FUNCTION_BLOCK FB 1051
TITLE = Blower PMP01
//Creation:
//Date:            Author:                                               Version
//--------------------------------------------------------------------------------
//29.03.2018     ilia                                   01.00.00
//
//Changes:
//No. Date:        Who       Description                           Mark   Version 
//--------------------------------------------------------------------------------
//01
//________________________________________________________________________________
//Function:
//1. Maximum 6 switching cycles per hour ' 10 minutes restart protection time
//
AUTHOR : ilia
NAME : project
VERSION : 1.0
VAR_INPUT
  IF_VP1_FC_DB : INT ;
  IF_VP1_FC_DW : INT ;
  i_piwPressureVP1 : INT ;	//analogue input address
  i_xSystemActive : BOOL ;	//system control on
  i_xFAValveClose : BOOL ;
  i_xFAValveOpen : BOOL ;
  ack_xFAValve : BOOL ;
  ack_OverPressureVP1 : BOOL ;
END_VAR
VAR_IN_OUT
  q_xFAValve : BOOL ;	//Fresh Air ventil
  f_xFAValve : BOOL ;	//Fault fresh air ventil
  f_xPressureFaultVP01 : BOOL ;	//Pressure Fault
  f_xBrokenWireVP01 : BOOL ;	//Broken wire pressure fault
  f_xParErrorVP01 : BOOL ;	//False parameter pressure transmitter
END_VAR
VAR
  reserve_IO : ARRAY  [10 .. 49 ] OF BYTE ;
  HMI : STRUCT 	//Interface of HMI
   CMD : STRUCT
    reserve : BOOL ;
    reserve_1 : BOOL ;
    reserve_2 : BOOL ;
    reserve_3 : BOOL ;
    reserve_4 : BOOL ;
    reserve_5 : BOOL ;
    reserve_6 : BOOL ;
    reserve_7 : BOOL ;
    reserve_8 : BOOL ;
    reserve_9 : BOOL ;
    reserve_10 : BOOL ;
    reserve_11 : BOOL ;
    reserve_12 : BOOL ;
    reserve_13 : BOOL ;
    reserve_14 : BOOL ;
    reserve_15 : BOOL ;
   END_STRUCT ;
   STATE : STRUCT
    xxPressureFault : BOOL ;
    xxEmtyPressure : BOOL ;
    xVP1Locked : BOOL ;
    reserve_4 : BOOL ;
    reserve_5 : BOOL ;
    reserve_6 : BOOL ;
    reserve_7 : BOOL ;
    reserve_8 : BOOL ;
    reserve_9 : BOOL ;
    reserve_10 : BOOL ;
    reserve_11 : BOOL ;
    reserve_12 : BOOL ;
    reserve_13 : BOOL ;
    reserve : BOOL ;
   END_STRUCT ;
   PARAM : STRUCT
    rOffDelayVPTime : REAL  := 6.000000e+001;
    rOnDelayHDTime : REAL ;
    res_1 : REAL ;
    res_2 : REAL ;
    res_3 : REAL ;
    res_4 : REAL  := 2.000000e+000;
    reserve_2 : REAL ;
    reserve_3 : REAL ;
    reserve_4 : INT ;
    reserve_4_1 : INT  := 6;
    reserve_6 : INT ;
    reserve_7 : INT ;
    reserve_8 : INT ;
    reserve_9 : INT ;
    reserve_9_1 : INT ;
   END_STRUCT ;
   PV : STRUCT
    rOffDelayVPTime : REAL ;
    rOnDelayHD : REAL ;
    rOffDelayRestart : REAL ;
    res : REAL ;
    res_1 : REAL ;
    res_2 : REAL ;
    res_3 : REAL ;
    res_4 : REAL ;
    reserve_4 : REAL ;
    reserve_8 : INT ;
    reserve_9 : INT ;
    reserve_10 : INT ;
    reserve_11 : INT ;
    reserve_8_1 : INT ;
   END_STRUCT ;
  END_STRUCT ;
  reserve_HMI : ARRAY  [146 .. 199 ] OF BYTE ;
  PROD : STRUCT 	//Interface of Production
   FROM : STRUCT
    reserve : INT ;
    reserve_1 : INT ;
    reserve_2 : INT ;
    reserve_3 : INT ;
    reserve_4 : INT ;
    reserve_5 : REAL ;
    reserve_6 : REAL ;
    CMD : STRUCT
     reserve : BOOL ;
     reserve_1 : BOOL ;
     reserve_2 : BOOL ;
     reserve_3 : BOOL ;
     reserve_4 : BOOL ;
     reserve_5 : BOOL ;
     reserve_6 : BOOL ;
     reserve_7 : BOOL ;
     reserve_8 : BOOL ;
     reserve_9 : BOOL ;
     reserve_10 : BOOL ;
     reserve_11 : BOOL ;
     reserve_12 : BOOL ;
     reserve_13 : BOOL ;
     reserve_14 : BOOL ;
     reserve_15 : BOOL ;
    END_STRUCT ;
   END_STRUCT ;
   TO : STRUCT
    reserve : INT ;
    reserve_1 : INT ;
    reserve_2 : INT ;
    reserve_3 : INT ;
    reserve_4 : INT ;
    reserve_5 : REAL ;
    reserve_6 : REAL ;
    STATE : STRUCT
     reserve : BOOL ;
     reserve_1 : BOOL ;
     reserve_2 : BOOL ;
     reserve_3 : BOOL ;
     reserve_4 : BOOL ;
     reserve_5 : BOOL ;
     reserve_6 : BOOL ;
     reserve_7 : BOOL ;
     reserve_8 : BOOL ;
     reserve_9 : BOOL ;
     reserve_10 : BOOL ;
     reserve_11 : BOOL ;
     reserve_12 : BOOL ;
     reserve_13 : BOOL ;
     reserve_14 : BOOL ;
     reserve_15 : BOOL ;
    END_STRUCT ;
   END_STRUCT ;
   reserve : ARRAY  [40 .. 49 ] OF BYTE ;
  END_STRUCT ;
  IF_Consumer : STRUCT 	//Interface Blower in blower object
   CONTROL : STRUCT
    Answer_DB : INT ;
    Answer_DW : INT ;
    iSpeedVP : INT ;
    reserve : INT ;
    reserve_3 : INT ;
    reserve_4 : REAL ;
    reserve_5 : REAL ;
    CMD : STRUCT
     xRequest : BOOL ;
     xRelease : BOOL ;
     reserve : BOOL ;
     reserve_1 : BOOL ;
     reserve_2 : BOOL ;
     reserve_3 : BOOL ;
     reserve_4 : BOOL ;
     reserve_5 : BOOL ;
     reserve_6 : BOOL ;
     reserve_7 : BOOL ;
     reserve_8 : BOOL ;
     reserve_9 : BOOL ;
     reserve_10 : BOOL ;
     reserve_11 : BOOL ;
     reserve_12 : BOOL ;
     reserve_13 : BOOL ;
    END_STRUCT ;
   END_STRUCT ;
   STATUS : STRUCT
    reserve_1 : INT ;
    reserve_2 : INT ;
    reserve_3 : INT ;
    reserve_4 : INT ;
    reserve_5 : INT ;
    rActualPressure : REAL ;
    reserve_6 : REAL ;
    STATE : STRUCT
     xReady : BOOL ;
     xActive : BOOL ;
     xPressureFault : BOOL ;
     xEmptyPressue : BOOL ;
     xFault : BOOL ;
     reserve : BOOL ;
     reserve_2 : BOOL ;
     reserve_3 : BOOL ;
     reserve_4 : BOOL ;
     reserve_5 : BOOL ;
     reserve_6 : BOOL ;
     reserve_7 : BOOL ;
     reserve_8 : BOOL ;
     reserve_9 : BOOL ;
     reserve_10 : BOOL ;
     reserve_11 : BOOL ;
    END_STRUCT ;
   END_STRUCT ;
  END_STRUCT ;
  IF_FC_VP1 : STRUCT 	//Interface FC in active object
   STATUS : STRUCT
    ActualFrequency : REAL ;
    reserve : INT ;
    reserve_1 : INT ;
    reserve_2 : INT ;
    reserve_3 : INT ;
    reserve_4 : INT ;
    reserve_5 : REAL ;
    STATE : STRUCT
     Ready : BOOL ;
     Active : BOOL ;
     Fault : BOOL ;
     reserve : BOOL ;
     reserve_1 : BOOL ;
     reserve_2 : BOOL ;
     reserve_3 : BOOL ;
     reserve_4 : BOOL ;
     reserve_5 : BOOL ;
     reserve_6 : BOOL ;
     reserve_7 : BOOL ;
     reserve_8 : BOOL ;
     reserve_9 : BOOL ;
     reserve_10 : BOOL ;
     reserve_11 : BOOL ;
     reserve_12 : BOOL ;
    END_STRUCT ;
   END_STRUCT ;
   CONTROL : STRUCT
    Answer_DB : INT ;
    Answer_DW : INT ;
    Frequency_Set : REAL ;
    No_motor_data : INT ;
    reserve : INT ;
    reserve_1 : INT ;
    reserve_2 : REAL ;
    CMD : STRUCT
     Request : BOOL ;
     Release : BOOL ;
     Left_run : BOOL ;
     reserve : BOOL ;
     reserve_1 : BOOL ;
     reserve_2 : BOOL ;
     reserve_3 : BOOL ;
     reserve_4 : BOOL ;
     reserve_5 : BOOL ;
     reserve_6 : BOOL ;
     reserve_7 : BOOL ;
     reserve_8 : BOOL ;
     reserve_9 : BOOL ;
     reserve_10 : BOOL ;
     reserve_11 : BOOL ;
     reserve_12 : BOOL ;
    END_STRUCT ;
   END_STRUCT ;
  END_STRUCT ;
  reserve_IF : ARRAY  [330 .. 499 ] OF BYTE ;
  VP1 : STRUCT 	//motor object
   parameter : STRUCT
    motor_on : BOOL  := TRUE;	//activate motor structure
    clock_on : BOOL ;	//activate clock structure
    FC_on : BOOL  := TRUE;	//activate frequency converter structure
    hour_meter_on : BOOL ;	//activate hour meter
    reserve_4 : BOOL ;
    reserve_5 : BOOL ;
    reserve_6 : BOOL ;
    reserve_7 : BOOL ;
   END_STRUCT ;
   quit_motor : BOOL ;	//1 = quit motor on
   input_motor : BOOL ;	//1 = input motor on (return indication)
   motor_locked : BOOL ;	//1 = motor locked (in manual and auto mode) e.g. repair-/safety switch
   auto_mode_control : BOOL ;	//1 = release/control of motor in auto mode
   motor_in_operation : BOOL ;	//1 = signal motor in operation
   fault : BOOL ;	//1 = signal motor fault
   man_mode_to_SCADA : BOOL ;	//0 = Automatik Mode, 1 = Hand Mode
   man_mode_from_SCADA : BOOL ;	//0 = Automatik Mode, 1 = Hand Mode
   man_mode_control : BOOL ;	//1 = release/control of motor in manual mode (from SCADA)
   man_mode_locked : BOOL ;	//1 = change to manual mode locked, motor is in automatic use
   start_with_impulse : BOOL  := TRUE;	//1 = start cycle with impulse
   set_cycles_reached : BOOL ;	//1 = set number of cycles has been reached
   continous_clock : BOOL  := TRUE;	//1 = continous clock / 0 = set number of clocks
   simulation : BOOL ;	//1 = simulation of object
   release_clock : BOOL ;	//1 = release bit for clock FC
   quit_clock : BOOL ;	//quit for clock FC, if release_clock = TRUE
   set_time_fault : INT  := 5;	//fault evaluation time in seconds
   actual_time_fault : INT ;	//actual fault evaluation time in seconds
   impulse_time : REAL  := 5.000000e+000;	//impulse time for clock in seconds
   break_time : REAL  := 5.000000e+000;	//break time for clock in seconds
   time_counter : REAL ;	//time counter (elapsed time)
   set_cycles : INT ;	//number of clocks if not continous clock
   clock_counter : INT ;	//clock counter
   FCs : STRUCT 	//frequency converter
    FC_in_operation : BOOL ;	//1 = FU in Betrieb
    fault : BOOL ;	//1 = FC fault
    set_revolutions_man_mode : INT  := 200;	//revolutions in permille in manual mode
    actual_revolutions : INT ;	//actual revolutions FC in man/auto mode
   END_STRUCT ;
   hour_meter : STRUCT 	//hour meter
    reset : BOOL ;	//reset hour meter
    warning : BOOL ;	//warning time exceeded
    alarm : BOOL ;	//alarm time exceeded
    actual_operating_hours : REAL ;	//actual operating hours (in hours)
    set_time_warning : REAL ;	//set time for warning (in hours)
    set_time_alarm : REAL ;	//set time for alarm (in hours)
    second_counter_oh : INT ;	//seconds of the actual operatin hours
   END_STRUCT ;
   system_on : BOOL ;	//system released resepectively system area released after emergency stopping
   object_state : INT ;	//1=grey; 5=green; 9=white; 15=yellow; 16=red
  END_STRUCT ;
  FAValve : STRUCT 	//Fresh Aur Valve object with 1Q and 0-2I
   parameter : STRUCT
    valve_on : BOOL  := TRUE;	//activate valve structure
    clock_on : BOOL ;	//activate clock structure
    reserve_3 : BOOL ;
    switching_number_on : BOOL ;	//activate switching number counter
    reserve_4 : BOOL ;
    parameter_1Q : BOOL ;	//valve type with 1 quit 0 inputs
    parameter_1Q_1I : BOOL ;	//valve type with 1 quit 1 input (=)
    parameter_1Q_1IN : BOOL ;	//valve type with 1 quit 1 input (<>)
    parameter_1Q_2I : BOOL  := TRUE;	//valve type with 1 quit 2 inputs
    parameter_text_pos_1 : BOOL ;
    parameter_text_straight : BOOL ;
    parameter_text_inverse : BOOL ;	//select text inverse = "close/open" or "bypass/convey" aso.
    parameter_text_open : BOOL ;	//select text quit = "open/close"
    parameter_text_convey : BOOL  := TRUE;	//select text quit = "convey/bypass"
    parameter_text_on : BOOL ;	//select text quit = "on/off"
    parameter_text_up : BOOL ;	//select text quit = "up/down"
   END_STRUCT ;
   quit_valve : BOOL ;	//1 = quit valve
   input_valve_set : BOOL ;	//1 = input valve, if quit valve set
   input_valve_not_set : BOOL ;	//1 = input valve, if quit valve not set
   auto_mode_control : BOOL ;	//1 = release/control of valve in auto mode
   valve_in_operation : BOOL ;	//1 = signal valve in operation
   fault : BOOL ;	//1 = signal valve fault
   man_mode_to_SCADA : BOOL ;	//0 = automatic mode , 1 = manual mode
   man_mode_from_SCADA : BOOL ;	//0 = automatic mode , 1 = manual mode
   man_mode_control : BOOL ;	//1 = release/control of valve in manual mode (from SCADA)
   man_mode_locked : BOOL ;	//1 = change to manual mode locked, valve is in automatic use
   start_with_impulse : BOOL ;	//1 = start cycle with impluse
   set_cycles_reached : BOOL ;	//1 = set number of cycles has been reached
   continous_clock : BOOL ;	//1 = continous clock / 0 = set number of clocks
   simulation : BOOL ;	//1 = simulation of object
   release_clock : BOOL ;	//1 = release bit for clock FC
   quit_clock : BOOL ;	//quit for clock FC, if release_clock = TRUE
   set_time_fault : INT  := 5;	//fault evaluation time in seconds
   actual_time_fault : INT ;	//actual fault evaluation time in seconds
   impulse_time : REAL  := 5.000000e+000;	//impulse time for clock in seconds
   break_time : REAL  := 5.000000e+000;	//break time for clock in seconds
   time_counter : REAL ;	//time counter (elapsed time)
   set_cycles : INT ;	//number of clocks if not continous clock
   clock_counter : INT ;	//clock counter
   switching_number_counter : STRUCT 	//switching number counter
    reset : BOOL ;	//reset switching number counter
    warning : BOOL ;	//warning number exceeded
    alarm : BOOL ;	//alarm number exceeded
    flank_flag : BOOL ;	//internal flag
    actual_switching_number : REAL ;	//actual switching number
    set_number_warning : REAL ;	//set number for warning
    set_number_alarm : REAL ;	//set number for alarm
   END_STRUCT ;
   set_time_in_operation : INT ;	//1IoO: set time for delay of "valve in operation"
   real_time_in_operation : INT ;	//1IoO: real time for delay of "valve in operation"
   system_on : BOOL ;	//system released resepectively system area released after emergency stopping
   reserve : ARRAY  [44 .. 47 ] OF BYTE ;
   object_state : INT ;	//1=grey; 5=green; 9=white; 15=yellow; 16=red
  END_STRUCT ;
  reserve_Cmod : ARRAY  [600 .. 999 ] OF BYTE ;
  PressureVP1 : STRUCT
   parameters : STRUCT
    pressureAIOn : BOOL  := TRUE;
    reserve1 : BOOL ;
    reserve2 : BOOL ;
    CounterOverPressure : BOOL  := TRUE;
    CounterEmptyPressure : BOOL ;
    CounterActivePressure : BOOL ;
    reserve_6 : BOOL ;
    reserve_7 : BOOL ;
    OverPressure : BOOL  := TRUE;
    EmptyPressure : BOOL  := TRUE;
    ActivePressure : BOOL  := TRUE;
    reserve_13 : BOOL ;
    ManOpSimEn : BOOL  := TRUE;
    ManOpAdjustEn : BOOL  := TRUE;
    reserve_14 : BOOL ;
    reserve_15 : BOOL ;
    uom_code : INT ;
   END_STRUCT ;
   ManModeAct : BOOL ;
   ManModeOp : BOOL ;
   ManModeLock : BOOL ;
   ManOpPressureEmpty : BOOL ;
   ManOpPressureConveying : BOOL ;
   ManOpPressureAlarm : BOOL ;
   ManOpPressureAdjust : BOOL ;
   SystemOn : BOOL ;
   ScalingErr : BOOL ;
   OVErr : BOOL ;
   ParErr : BOOL ;
   fOverPressure : BOOL ;
   fOverPressureEn : BOOL ;
   fOverPressureAck : BOOL ;
   Overpressure : BOOL ;
   EmptyPressure : BOOL ;
   ActivePressure : BOOL ;
   Active : BOOL ;
   AdjustRelease : BOOL ;
   AdjustPulse : BOOL ;
   ManAdjustReq : BOOL ;
   ManAdjustRdy : BOOL ;
   CounterReset : BOOL ;
   CounterEdge : BOOL ;
   PVAct : REAL ;
   PressureOffset : REAL ;
   MaxOverPressurePV : REAL  := -6.000000e+002;
   MinOverPressurePV : REAL  := -3.000000e+002;
   EmptyPressurePV : REAL  := -2.000000e+002;
   ActivePressurePV : REAL ;
   EmptyDelay : INT  := 5;
   ActiveDelay : INT  := 5;
   AlarmDelay : INT  := 10;
   EmptyDelayCounter : INT ;
   ActiveDelayCounter : INT ;
   AlarmDelayCounter : INT ;
   CounterAct : REAL ;
   object_state : INT ;
  END_STRUCT ;
  reserve_Binary : ARRAY  [1050 .. 1499 ] OF BYTE ;
  TIMES : STRUCT 	//ten timers
   TOF_DelayVP : STRUCT
    IN : BOOL ;
    RST : BOOL ;
    IMP : BOOL ;
    Q : BOOL ;
    PT : REAL ;
    ET : REAL ;
   END_STRUCT ;
   TOF_RestartProtectVP1 : STRUCT
    IN : BOOL ;
    RST : BOOL ;
    IMP : BOOL ;
    Q : BOOL ;
    PT : REAL ;
    ET : REAL ;
   END_STRUCT ;
   TON_HoseDiverter : STRUCT
    IN : BOOL ;
    RST : BOOL ;
    IMP : BOOL ;
    Q : BOOL ;
    PT : REAL  := 2.000000e+000;
    ET : REAL ;
   END_STRUCT ;
   TOF_HoseDiverter : STRUCT
    IN : BOOL ;
    RST : BOOL ;
    IMP : BOOL ;
    Q : BOOL ;
    PT : REAL ;
    ET : REAL ;
   END_STRUCT ;
   reserve_3 : STRUCT
    IN : BOOL ;
    RST : BOOL ;
    IMP : BOOL ;
    Q : BOOL ;
    PT : REAL ;
    ET : REAL ;
   END_STRUCT ;
   reserve_4 : STRUCT
    IN : BOOL ;
    RST : BOOL ;
    IMP : BOOL ;
    Q : BOOL ;
    PT : REAL ;
    ET : REAL ;
   END_STRUCT ;
   reserve_5 : STRUCT
    IN : BOOL ;
    RST : BOOL ;
    IMP : BOOL ;
    Q : BOOL ;
    PT : REAL ;
    ET : REAL ;
   END_STRUCT ;
   reserve_6 : STRUCT
    IN : BOOL ;
    RST : BOOL ;
    IMP : BOOL ;
    Q : BOOL ;
    PT : REAL ;
    ET : REAL ;
   END_STRUCT ;
  END_STRUCT ;
  SEQUENCES : STRUCT
   Sequence : STRUCT
    AUTO : BOOL ;
    MANUAL : BOOL ;
    LOCKED : BOOL ;
    RELEASE : BOOL ;
    ACTIVE : BOOL ;
    reserve_2 : BOOL ;
    reserve_3 : BOOL ;
    reserve_4 : BOOL ;
    reserve_5 : BOOL ;
    reserve_6 : BOOL ;
    reserve_7 : BOOL ;
    reserve_8 : BOOL ;
    reserve_9 : BOOL ;
    reserve_10 : BOOL ;
    reserve_11 : BOOL ;
    reserve_12 : BOOL ;
   END_STRUCT ;
   reserve : ARRAY  [2 .. 99 ] OF BYTE ;
  END_STRUCT ;
  INTERNAL : STRUCT
   IF : STRUCT
    VacuumPump : STRUCT
     VP1_FaultControl : BOOL ;
     VP2_FaultControl : BOOL ;
     reserve : BOOL ;
     reserve_2 : BOOL ;
     reserve_3 : BOOL ;
     reserve_4 : BOOL ;
     reserve_5 : BOOL ;
     reserve_5_1 : BOOL ;
     SpeedVP1_PARAM : INT ;
     SpeedVP1_PV : REAL ;
    END_STRUCT ;
    SF01 : STRUCT
     HighLevelSF_FaultControl : BOOL ;
     ManFlapSF_FaultControl : BOOL ;
     SF_ready : BOOL ;
     CleaningFilterAfterSeq : BOOL ;
     reserve : BOOL ;
     resrve : BOOL ;
     res : BOOL ;
     res_1 : BOOL ;
     res_2 : INT ;
     res_3 : REAL ;
    END_STRUCT ;
    VP_FC : STRUCT
     free : BOOL ;
     res_2 : BOOL ;
     res_3 : BOOL ;
     res_4 : BOOL ;
     reserve : BOOL ;
     resrve : BOOL ;
     res : BOOL ;
     res_1 : BOOL ;
    END_STRUCT ;
    reserve_6 : BOOL ;
    reserve_7 : BOOL ;
    reserve_8 : BOOL ;
    reserve_9 : BOOL ;
    reserve_10 : BOOL ;
    reserve_11 : BOOL ;
    reserve_12 : BOOL ;
    reserve_13 : BOOL ;
    reserve_14 : BOOL ;
    reserve_15 : BOOL ;
   END_STRUCT ;
   Flags : STRUCT
    BinaryObjects : STRUCT
     Res : BOOL ;
     Res_1 : BOOL ;
     RES_2 : BOOL ;
     RES_3 : BOOL ;
     RES_4 : BOOL ;
     RES_5 : BOOL ;
     RES_6 : BOOL ;
     RES_7 : BOOL ;
    END_STRUCT ;
    FP_VP1_ON : STRUCT
     help : BOOL ;
     pulse : BOOL ;
    END_STRUCT ;
    Res_1 : STRUCT
     help : BOOL ;
     pulse : BOOL ;
    END_STRUCT ;
    FN_SequenceActive : STRUCT
     help : BOOL ;
     pulse : BOOL ;
    END_STRUCT ;
    FP_reserve : STRUCT
     help : BOOL ;
     pulse : BOOL ;
    END_STRUCT ;
    reserve_3 : BOOL ;
    reserve_4 : BOOL ;
    reserve_5 : BOOL ;
    reserve_6 : BOOL ;
    reserve_7 : BOOL ;
    reserve_8 : BOOL ;
    reserve_9 : BOOL ;
    reserve_10 : BOOL ;
   END_STRUCT ;
   PressureTransmitter : STRUCT
    Analog : STRUCT
     in : STRUCT
      UperLimit : REAL  := 1.000000e+003;	//Uper limit analog value
      LowerLimit : REAL  := -1.000000e+003;	//Lower limit analog value
      MaxDigit : REAL  := 2.764800e+004;	//Uper limit analog channel
      MinDigit : REAL ;	//Lower limit analog channel
      Simulation : BOOL ;	//Simulation = 1
      DB_Simulation_IO : INT  := 92;	//DB for simulation
     END_STRUCT ;
     out : STRUCT
      Value : REAL ;	//IO Analog value
      Broken_wire : BOOL ;	//Fault broken wire
      Reserve : INT ;
     END_STRUCT ;
    END_STRUCT ;
    Evaluation : STRUCT
     in : STRUCT
      Delay_Adjust : REAL  := 1.000000e+001;	//Delay adjust of Pressure Transmitter
      Selection_S_D : CHAR  := 'S';	//Selection suction-/pressure conveying ('S' or 'D')
      REL_Pressure_fault : BOOL  := TRUE;	//Release Pressure fault
      Time_counter : REAL ;	//Time counter delay adjust
      Output_Timer : BOOL ;	//Timer output delay adjust
     END_STRUCT ;
     out : STRUCT
      Relative_Pressure : REAL ;	//Relative Pressure
      Memory_Pressure : REAL ;	//Memory Pressure
      Pressure_fault_active : BOOL ;	//Pressure fault
      Empty_Pressure_reached : BOOL ;	//Below Empty Pressure
      output_delay_calibration : BOOL ;
     END_STRUCT ;
    END_STRUCT ;
   END_STRUCT ;
   Instance_DB_number : INT ;
   RestartProtectTime : REAL ;
  END_STRUCT ;
END_VAR
VAR_TEMP
  dummyBool : BOOL ;
END_VAR
BEGIN
NETWORK
TITLE = ---- instance DB ----
      L     0;
      L     DINO;
      ==I;
      BEC;
      T     #INTERNAL.Instance_DB_number;
NETWORK
TITLE = ----------------SEQUENCES AUTO/LOCKED/MANUAL-----------------
NETWORK
TITLE =  Sequence AUTO
      AN    #SEQUENCES.Sequence.LOCKED;
      =     #SEQUENCES.Sequence.AUTO;
NETWORK
TITLE =  Sequence Manual
      O     #VP1.man_mode_to_SCADA;
      O     #FAValve.man_mode_to_SCADA;
      =     #SEQUENCES.Sequence.MANUAL;
NETWORK
TITLE =  Sequence Locked
//BLOCK VP ALSO??????
      A     #SEQUENCES.Sequence.MANUAL;
      ON    #i_xSystemActive;
// MUST BE BLOCK VP 
      =     #SEQUENCES.Sequence.LOCKED;
NETWORK
TITLE = ---------------------SENSORS/SWITCHES --------------------------
NETWORK
TITLE = ------------------PRESSURE TRANSMITTERS-------------------------
NETWORK
TITLE = PressureTransmitter VP01
      L     -5.000000e+00;	// 2.000000e+001 
      T     #PressureVP1.ActivePressurePV;
      CALL  FC 29 (
           ManOpEn                  := TRUE,
           ManModeTrack             := TRUE,
           NegEvalEn                := TRUE,
           OVErrEn                  := TRUE,
           AlarmOprEn               := TRUE,
           AlarmOprAckEn            := FALSE,
           DigitMin                 := 0,
           DigitMax                 := 27648,
           ValueMin                 := -1.000000e+03,
           ValueMax                 := 1.000000e+03,
           ValueSubs                := 1.000000e+01,
           Configuration            := W#16#0,
           UOM                      := 1138,
           iSystemOn                := #i_xSystemActive,
           iwDigit                  := #i_piwPressureVP1,
           iActive                  := #PressureVP1.Active,
           aAlarmOprAck             := #ack_OverPressureVP1,
           PVAct                    := #PressureVP1.PVAct,
           fAlarmOpr                := #PressureVP1.fOverPressure,
           OverPressure             := #PressureVP1.Overpressure,
           EmptyPressure            := #PressureVP1.EmptyPressure,
           ActivePressure           := #PressureVP1.ActivePressure,
           fScalingErr              := #PressureVP1.ScalingErr,
           fOVErr                   := #PressureVP1.OVErr,
           fParErr                  := #f_xParErrorVP01,
           ioStructure              := #PressureVP1);	//mbar / #fPressureFault
      A     #PressureVP1.fOverPressure;	// #PressureTransmittter.Overpressure
      =     #f_xPressureFaultVP01;
      A     #PressureVP1.OVErr;
      =     #f_xBrokenWireVP01;
NETWORK
TITLE = -----------------------------SEQUENCES--------------------------
NETWORK
TITLE = Sequence: ready to consumer
      A     #SEQUENCES.Sequence.AUTO;
      A     #IF_Consumer.CONTROL.CMD.xRequest;
      AN    #f_xFAValve;
      =     #IF_Consumer.STATUS.STATE.xReady;
NETWORK
TITLE = Sequence: release vacuum pump (VP1)
//blower off delay
      A     #SEQUENCES.Sequence.AUTO;
      A     #IF_Consumer.CONTROL.CMD.xRequest;
      A     #IF_Consumer.STATUS.STATE.xReady;
      A     #IF_Consumer.CONTROL.CMD.xRelease;
      =     #TIMES.TOF_DelayVP.IN;
      ON    #i_xSystemActive;
      =     #TIMES.TOF_DelayVP.RST;
      CALL  FC 3 (
           in_Freigabe              := #TIMES.TOF_DelayVP.IN,
           in_Reset                 := #TIMES.TOF_DelayVP.RST,
           in_Impuls                := M 1.7,
           in_Impulszeit_in_100ms   := MW 6,
           in_Verzoegerungsart      := B#16#41,
           in_Verzoegerungszeit     := #HMI.PARAM.rOffDelayVPTime,
           io_Ausgangssignal        := #TIMES.TOF_DelayVP.Q,
           io_Zeitzaehler           := #TIMES.TOF_DelayVP.ET);
      L     #TIMES.TOF_DelayVP.ET;
      T     #HMI.PV.rOffDelayVPTime;
      A     #TIMES.TOF_DelayVP.Q;
      =     #VP1.auto_mode_control;
NETWORK
TITLE = Sequence: release VP1 - with frequency Converter
//FC request
      A     #SEQUENCES.Sequence.AUTO;
      A     #IF_Consumer.CONTROL.CMD.xRequest;
      A     #IF_Consumer.STATUS.STATE.xReady;
      O;
      A     #VP1.man_mode_to_SCADA;
      A     #VP1.man_mode_control;
      O;
      A     #IF_FC_VP1.STATUS.STATE.Active;
      =     #IF_FC_VP1.CONTROL.CMD.Request;
      A     #TIMES.TOF_RestartProtectVP1.Q;
      AN    #VP1.motor_in_operation;
      O;
      AN    #IF_FC_VP1.STATUS.STATE.Ready;
      A     #IF_FC_VP1.CONTROL.CMD.Request;
      O;
      A     #IF_FC_VP1.STATUS.STATE.Fault;
      =     #VP1.motor_locked;
      A     #VP1.quit_motor;
      =     #VP1.input_motor;
      CALL  FC 20 (
           in_Handbedienung_erlaubt := TRUE,
           in_Quitt_Stoerung_noetig := TRUE,
           in_Anlage_ein            := #i_xSystemActive,
           in_Quitt_Stoerung        := #dummyBool,
           in_Ansteuerung_Motor     := #VP1.auto_mode_control,
           in_Eingang_Motor         := #VP1.input_motor,
           io_Ausgang_Motor         := #VP1.quit_motor,
           io_Motor_in_Betrieb      := #VP1.motor_in_operation,
           io_Stoerung              := #VP1.fault,
           io_Motorstruktur         := #VP1);
//FC release
      A(;
      A     #VP1.auto_mode_control;
      O;
      A     #VP1.man_mode_to_SCADA;
      A     #VP1.man_mode_control;
      );
      A     #IF_FC_VP1.CONTROL.CMD.Request;
      A     #IF_FC_VP1.STATUS.STATE.Ready;
      A     #VP1.motor_in_operation;
      =     #IF_FC_VP1.CONTROL.CMD.Release;
NETWORK
TITLE = Sequence: frequency to/from FC VP1
      A     #VP1.man_mode_to_SCADA;
      A     #VP1.man_mode_control;
      L     #IF_Consumer.CONTROL.iSpeedVP;
      JCN   VNM;	// man mode 
      L     #VP1.FCs.set_revolutions_man_mode;
      L     10;
      /I;
VNM:  T     #INTERNAL.IF.VacuumPump.SpeedVP1_PARAM;
// to FC
      L     #INTERNAL.IF.VacuumPump.SpeedVP1_PARAM;
      ITD;
      DTR;
      T     #IF_FC_VP1.CONTROL.Frequency_Set;
//from FC
      L     #IF_FC_VP1.STATUS.ActualFrequency;
      T     #INTERNAL.IF.VacuumPump.SpeedVP1_PV;
      A     #VP1.man_mode_to_SCADA;
      A     #VP1.man_mode_control;
      L     0;
      JCN   VNM1;
      L     #INTERNAL.IF.VacuumPump.SpeedVP1_PV;
      RND;
      L     10;
      *I;
VNM1: T     #VP1.FCs.actual_revolutions;
NETWORK
TITLE = Sequence: Restart VP1 Protection
//only 12 times per hour
// >>test 30.0 sek, for production 300.0 sek
      L     3.000000e+02;
      T     #INTERNAL.RestartProtectTime;
//<<tests
//restart protection 
      A     #IF_FC_VP1.STATUS.STATE.Active;
      A     #VP1.motor_in_operation;
      FP    #INTERNAL.Flags.FP_VP1_ON.help;
      =     #TIMES.TOF_RestartProtectVP1.IN;
      CALL  FC 3 (
           in_Freigabe              := #TIMES.TOF_RestartProtectVP1.IN,
           in_Reset                 := FALSE,
           in_Impuls                := M 1.7,
           in_Impulszeit_in_100ms   := MW 6,
           in_Verzoegerungsart      := B#16#41,
           in_Verzoegerungszeit     := #INTERNAL.RestartProtectTime,
           io_Ausgangssignal        := #TIMES.TOF_RestartProtectVP1.Q,
           io_Zeitzaehler           := #TIMES.TOF_RestartProtectVP1.ET);
      L     #TIMES.TOF_RestartProtectVP1.ET;
      T     #HMI.PV.rOffDelayRestart;
      L     #TIMES.TOF_RestartProtectVP1.ET;
      T     #HMI.PV.rOffDelayRestart;
NETWORK
TITLE = Sequence: control fresh air valve
      A     #SEQUENCES.Sequence.AUTO;
      A     #VP1.motor_in_operation;
      =     #TIMES.TON_HoseDiverter.IN;
      AN    #i_xSystemActive;
      =     #TIMES.TON_HoseDiverter.RST;
      CALL  FC 3 (
           in_Freigabe              := #TIMES.TON_HoseDiverter.IN,
           in_Reset                 := #TIMES.TON_HoseDiverter.RST,
           in_Impuls                := M 1.7,
           in_Impulszeit_in_100ms   := MW 6,
           in_Verzoegerungsart      := B#16#45,
           in_Verzoegerungszeit     := 3.000000e+00,
           io_Ausgangssignal        := #TIMES.TON_HoseDiverter.Q,
           io_Zeitzaehler           := #TIMES.TON_HoseDiverter.ET);
      A     #TIMES.TON_HoseDiverter.Q;
      =     #FAValve.auto_mode_control;
NETWORK
TITLE = Sequence: statuses to consumer
      A     #SEQUENCES.Sequence.AUTO;
      A     #IF_Consumer.CONTROL.CMD.xRelease;
      A     #VP1.motor_in_operation;
      A     #IF_FC_VP1.STATUS.STATE.Active;
      A     #FAValve.valve_in_operation;
      =     #SEQUENCES.Sequence.ACTIVE;
      A     #SEQUENCES.Sequence.ACTIVE;
      A     #IF_Consumer.STATUS.STATE.xReady;
      A     #IF_Consumer.CONTROL.CMD.xRelease;
      =     #IF_Consumer.STATUS.STATE.xActive;
//pressure fault
//emty pressure reached
//actual pressure 
      L     #PressureVP1.PVAct;
//  L     -5.100000e+002
      T     #IF_Consumer.STATUS.rActualPressure;
      O     #VP1.fault;
      O     #IF_FC_VP1.STATUS.STATE.Fault;
      O     #FAValve.fault;
      O     #PressureVP1.OVErr;
      =     #IF_Consumer.STATUS.STATE.xFault;
NETWORK
TITLE = Call fresh air Valve
      CALL  FC 21 (
           in_Ventil_Typ            := 1,
           in_Handbedienung_erlaubt := TRUE,
           in_Quitt_Stoerung_noetig := FALSE,
           in_Quitt_Stoerung        := TRUE,
           in_Anlage_ein            := #i_xSystemActive,
           in_Ansteuerung_Ventil    := #FAValve.auto_mode_control,
           in_Eingang_angesteuert   := #i_xFAValveClose,
           in_Eingang_nicht_angest  := #i_xFAValveOpen,
           io_Ausgang_Ventil        := #q_xFAValve,
           io_Ventil_in_Betrieb     := #FAValve.valve_in_operation,
           io_Stoerung              := #f_xFAValve,
           io_Ventilstruktur        := #FAValve);	// service mode available from plc /  ack needed
      A     #FAValve.man_mode_control;
      =     #FAValve.man_mode_control;
NETWORK
TITLE = -------------------STATUS TO HMI--------------------------------
NETWORK
TITLE = Sequence: Restart block to HMI
      A     #TIMES.TOF_RestartProtectVP1.Q;
      AN    #VP1.motor_in_operation;
      =     #HMI.STATE.xVP1Locked;
NETWORK
TITLE = ---- Interface ----
NETWORK
TITLE = interface FC
      CALL  FC 40 (
           i_Freigabe               := #IF_FC_VP1.CONTROL.CMD.Request,
           i_Ziel_DB                := #IF_VP1_FC_DB,
           i_Ziel_DW                := #IF_VP1_FC_DW,
           i_SST_von_Ziel           := #IF_FC_VP1.STATUS,
           i_SST_an_Ziel            := #IF_FC_VP1.CONTROL,
           Ziel_frei                := #INTERNAL.IF.VP_FC.free);
NETWORK
TITLE = interface Consumer
      CALL  FC 41 (
           i_SST_von_Ziel           := #IF_Consumer.CONTROL,
           i_SST_an_Ziel            := #IF_Consumer.STATUS);
END_FUNCTION_BLOCK

FUNCTION_BLOCK FB 4900
TITLE = Call Frequency Converters
//Creation:
//Date:            Author:                                               Version
//--------------------------------------------------------------------------------
//29.03.2018        ilia                                                 01.00.00
//
//Changes:
//No. Date:        Who       Description                           Mark   Version 
//--------------------------------------------------------------------------------
//01
//________________________________________________________________________________
//Function:
AUTHOR : ilia
NAME : project
VERSION : 1.0
BEGIN
NETWORK
TITLE = Vacuum Pump VP01
      CALL  FB 4901 , DB 10001 (
           in_FU_Typ                := 6,
           in_PEA_Adresse           := 1000,
           in_FU_Nummer             := 1,
           in_Motornennfrequenz     := 5.000000e+01,
           in_Motornenndrehzahl     := 1.455000e+03,
           aFU                      := DB35.DBX 200.0,
           FU_Stoerung              := DB34.DBX 200.0);	//1.455000e+003
END_FUNCTION_BLOCK

FUNCTION_BLOCK FB 4901
TITLE = FU Auswahlbaustein
//Erstellung:
//Datum        Bearbeiter                                                 Version
//--------------------------------------------------------------------------------
//10.07.06     Dominik Ilzhöfer (id)                                      01.00.00
//
//Änderungen:
//Nr. Datum    Bearb Änderung                                       Marke  Version
//--------------------------------------------------------------------------------
//01  06.11.07 sra   Motornennfrequenz und Motornenndrehzahl eingef.(001) 01.01.00
//02  23.07.13 sra   Status FU eingefügt                            (002) 01.02.00
//
//Baustein zur Ansteuerung von Frequenzumformern über Profibus-DB
//
//Parametrierung:
//FU-Typ:        wird zur richtigen Fehleranzeige an der Visualisierung benötigt
//               1=Siemens-MM4
//               2=SEW UFP11A
//               3=Lenze E82ZAFPC
//               4=Danfoss VLT5000
//               5=Danfoss FC300
//               6=SEW DFP21B
//             
//PEA-Adresse:   Anfangsadresse der Profibus-Schnittstelle
//Motordaten-DB: DB-Nummer mit Motordaten (Standard = DB4)
//FU-Nummer    : wird nur bei SEW Frequenzumformern mit UFP11A und DFP21B benötigt
//
//!Achtung!
//Bei den SEW Frequenzumformern wird die Motornennfrequenz und die 
//Motornenndrehzahl benötigt. D.h. es muss entweder ein Motordatensatz in dem 
//Motordaten-DB vorhanden sein oder die Werte müssen dem Baustein übergeben 
//werden.
NAME : standard
VERSION : 1.2
VAR_INPUT
  in_FU_Typ : INT ;	//1=Siemens-MM4, 2=SEW UFP11A, 3=Lenze E82ZAFPC, 4=Danfoss VLT5000
  in_PEA_Adresse : INT ;	//Basisadresse für EA-Daten im PEA-Bereich
  in_Motordaten_DB : INT  := 1;	//Adresse des DBs für Motordaten ( 0 = keine Motordaten schreiben )
  in_FU_Nummer : INT ;	//Nummer des FUs (für SEW-FUs)
  in_Motornennfrequenz : REAL ;	//muss bei SEW-FUs angegeben werden wenn kein Motordatensatz vorhanden ist
  in_Motornenndrehzahl : REAL ;	//muss bei SEW-FUs angegeben werden wenn kein Motordatensatz vorhanden ist
  aFU : BOOL ;
END_VAR
VAR_IN_OUT
  FU_Stoerung : BOOL ;
END_VAR
VAR
  reserve : ARRAY  [20 .. 29 ] OF BYTE ;
  Daten_Visualisierung : STRUCT
   von : STRUCT
    Quittierung_Stoerung : BOOL ;
    reserve : ARRAY  [2 .. 19 ] OF BYTE ;
   END_STRUCT ;
   an : STRUCT
    FU_Typ : INT ;
    Freigabe : BOOL ;
    Laeuft : BOOL ;
    Stoerung : BOOL ;
    Warnung : BOOL ;
    Sollfrequenz_erreicht : BOOL ;
    Sollfrequenz : REAL ;
    Istfrequenz : REAL ;
    Istdrehzahl : REAL ;
    Ausgangsstrom : REAL ;
    Leistung : REAL ;
    Drehmoment : REAL ;
    Spannung : REAL ;
    FU_Nummer : INT ;
    FB_Fehlermeldung : INT ;
    Stoerungsnummer : DINT ;
    reserve : ARRAY  [40 .. 47 ] OF BYTE ;
    Status : INT ;
   END_STRUCT ;
  END_STRUCT ;
  Schnittstelle : STRUCT
   von : STRUCT
    Antwort_DB : INT ;
    Antwort_DW : INT ;
    Sollfrequenz : REAL ;
    Motordatensatz_Nummer : INT ;
    reserve : ARRAY  [10 .. 17 ] OF BYTE ;
    Steuerbits : STRUCT
     Anforderung : BOOL ;
     Freigabe : BOOL ;
     Linkslauf : BOOL ;
    END_STRUCT ;
   END_STRUCT ;
   an : STRUCT
    Istfrequenz : REAL ;
    reserve : ARRAY  [4 .. 17 ] OF BYTE ;
    Statusbits : STRUCT
     Bereit : BOOL ;
     Laeuft : BOOL ;
     Stoerung : BOOL ;
    END_STRUCT ;
   END_STRUCT ;
  END_STRUCT ;
  Motordaten : STRUCT
   Nennleistugsfaktor : REAL ;
   Nennfrequenz : REAL ;
   Nenndrehzahl : REAL ;
   Nennstrom : REAL ;
   Nennspannung : REAL ;
   Nennleistung : REAL ;
   reserve : ARRAY  [24 .. 29 ] OF BYTE ;
  END_STRUCT ;
  Profibus_FB : FB 6119;
END_VAR
VAR_TEMP
  Motordaten_schreiben : BOOL ;
  Motordaten_Transfer_Fehl : INT ;
  Motordaten_Adresse_Quell : INT ;
  Motordaten_Adresse_Ziel : INT ;
END_VAR
BEGIN
NETWORK
TITLE = "Motordaten_schreiben" bilden
//Motordaten werden nur geschrieben, wenn ein Motordaten_DB und eine 
//Motordatensatz_Nummer ungleich 0 angegeben werden
      A(;
      L     #in_Motordaten_DB;
      L     0;
      <>I;
      );
      A(;
      L     #Schnittstelle.von.Motordatensatz_Nummer;
      L     0;
      <>I;
      );
      =     #Motordaten_schreiben;
NETWORK
TITLE = Motordatensatz in Motordaten kopieren
//Kompletter Motordatensatz wird aus Motordaten_DB kopiert
      L     #in_Motornennfrequenz;	// (001)
      T     #Motordaten.Nennfrequenz;	// (001)
      L     #in_Motornenndrehzahl;	// (001)
      T     #Motordaten.Nenndrehzahl;	// (001)
      A     #Motordaten_schreiben;
      JCN   SPR1;
      L     #Schnittstelle.von.Motordatensatz_Nummer;	// Nummer des Datensatzes des Motors
      L     -1;
      +I;
      L     30;	// Länge eines Datensatzes
      *I;
      T     #Motordaten_Adresse_Quell;	// Anfangsadresse des Datensatzes
      L     P##Motordaten;
      SRD   3;
      T     #Motordaten_Adresse_Ziel;
      CALL  FC 5 (
           Quell_Typ                := B#16#44,
           Quell_DB                 := #in_Motordaten_DB,
           Quell_DW                 := #Motordaten_Adresse_Quell,
           Ziel_Typ                 := B#16#49,
           Ziel_DB                  := 0,
           Ziel_DW                  := #Motordaten_Adresse_Ziel,
           Block_Laenge             := 24,
           outFehler                := #Motordaten_Transfer_Fehl);	// DB mit den Motordatensätzen /  Anfangsadresse des Datensatzes /  nicht verwendet da Ziel_Typ :='I' /  Abhängig vom Motordaten_DB
SPR1: NOP   0;
NETWORK
TITLE = Bei Anforderung "Bereit" bilden
      A     #Schnittstelle.von.Steuerbits.Anforderung;
      =     #Schnittstelle.an.Statusbits.Bereit;
NETWORK
TITLE = Auswahl des FU-Typs
//In der Multiinstanz "Profibus_FB" benötigten FU_Baustein im Datentyp angeben
      CALL  #Profibus_FB (
           in_PEA_Adresse           := #in_PEA_Adresse,
           in_FU_Nummer             := #in_FU_Nummer,
           in_Motordaten_J_N        := #Motordaten_schreiben,
           in_Freigabe              := #Schnittstelle.von.Steuerbits.Freigabe,
           in_Linkslauf             := #Schnittstelle.von.Steuerbits.Linkslauf,
           in_Quittierung_Stoerung  := #Daten_Visualisierung.von.Quittierung_Stoerung,
           in_Sollfrequenz          := #Schnittstelle.von.Sollfrequenz,
           in_Motorleistungsfaktor  := #Motordaten.Nennleistugsfaktor,
           in_Motornennfrequenz     := #Motordaten.Nennfrequenz,
           in_Motornenndrehzahl     := #Motordaten.Nenndrehzahl,
           in_Motornennstrom        := #Motordaten.Nennstrom,
           in_Motornennspannung     := #Motordaten.Nennspannung,
           in_Motornennleistung     := #Motordaten.Nennleistung,
           out_Istfrequenz          := #Daten_Visualisierung.an.Istfrequenz,
           out_Istdrehzahl          := #Daten_Visualisierung.an.Istdrehzahl,
           out_Leistung             := #Daten_Visualisierung.an.Leistung,
           out_Drehmoment           := #Daten_Visualisierung.an.Drehmoment,
           out_Motorspannung        := #Daten_Visualisierung.an.Spannung,
           out_Ausgangsstrom        := #Daten_Visualisierung.an.Ausgangsstrom,
           out_Stoerung             := #Daten_Visualisierung.an.Stoerung,
           out_Warnung              := #Daten_Visualisierung.an.Warnung,
           out_Sollwert_erreicht    := #Daten_Visualisierung.an.Sollfrequenz_erreicht,
           out_laeuft               := #Daten_Visualisierung.an.Laeuft,
           out_FB_Fehlermeldung     := #Daten_Visualisierung.an.FB_Fehlermeldung,
           out_Stoerungsnummer      := #Daten_Visualisierung.an.Stoerungsnummer);
NETWORK
TITLE = Verknüpfungen von Signalen für Visu und Schnittstelle
      L     #in_FU_Typ;
      T     #Daten_Visualisierung.an.FU_Typ;
      L     #in_FU_Nummer;
      T     #Daten_Visualisierung.an.FU_Nummer;
      A     #Schnittstelle.von.Steuerbits.Freigabe;
      =     #Daten_Visualisierung.an.Freigabe;
      L     #Schnittstelle.von.Sollfrequenz;
      T     #Daten_Visualisierung.an.Sollfrequenz;
      L     #Daten_Visualisierung.an.Istfrequenz;
      T     #Schnittstelle.an.Istfrequenz;
      A     #Daten_Visualisierung.an.Laeuft;
      =     #Schnittstelle.an.Statusbits.Laeuft;
      A     #Daten_Visualisierung.an.Stoerung;
      =     #Schnittstelle.an.Statusbits.Stoerung;
      =     #FU_Stoerung;
NETWORK
TITLE = Sollfrequenz löschen
      A     #Schnittstelle.von.Steuerbits.Freigabe;
      JC    M001;
      L     0;
      T     #Schnittstelle.von.Sollfrequenz;
      CLR;
      =     #Daten_Visualisierung.an.Sollfrequenz_erreicht;
M001: NOP   0;
NETWORK
TITLE = Statusanzeige für Visualisierung
//(002)
      L     16;	// Status Störung
      A     #Daten_Visualisierung.an.Stoerung;
      JC    Stat;
      L     13;	// Status Warnung
      A     #Daten_Visualisierung.an.Warnung;
      JC    Stat;
      L     5;	// Status läuft
      A     #Daten_Visualisierung.an.Laeuft;
      JC    Stat;
      L     1;	// Status aus
Stat: T     #Daten_Visualisierung.an.Status;
NETWORK
TITLE = Acknowledge FU Fault from the Visualization 
      A     #aFU;
      =     #Daten_Visualisierung.von.Quittierung_Stoerung;
NETWORK
TITLE = Schnittstellendaten kopieren
      CALL  FC 41 (
           i_SST_von_Ziel           := #Schnittstelle.von,
           i_SST_an_Ziel            := #Schnittstelle.an);
END_FUNCTION_BLOCK

FUNCTION_BLOCK FB 6119
TITLE = Control of SEW frequency converter with DFE32B via Profinet
//Building:
//Date         Editor                                                     Version
//--------------------------------------------------------------------------------
//31.08.10     A.Kremer (kal)                                            01.00.00
//
//Modifications:
//No. Date     Edit  Description                                    Index Version
//--------------------------------------------------------------------------------
//01  24.04.12 sra   Anpassung zur Integration als Standardbaustein (001) 01.01.00
//02  23.11.15 kst   Anpassung allgemein                            (002) 01.02.00
//03  17.02.16 sra   out_FB_Fehlermeldung = INT                     (003) 01.02.01
//________________________________________________________________________________
//Functional description:
//
//The function cummunicates to a SEW frequency converter MOVITRAC B via Profinet
//interface DFE32B.
//
//Hardwareconfiguration:
//Install GSDML file in hardware catalogue:
// GSDML-V2.1-SEW-DFE-DFS-2Ports-20070426.xml (Internet: www.SEW-EURODRIVE.de)
//
//After the installation you can find the Profinet module  "SEW Gateway DFE32B 
//V1.2" in the hardware catalogue under the menu: "Profinet IO -> other FIELD 
//DEVICES -> Drives -> SEW -> DFE/DFS (2Ports) ->"
//
//Insert this module to the hardware and configurate the following module
//     Slot 1: Empty
//from Slot 2: AS 1 Antrieb (1x3PD)   as often as the number of freq.converter    
// 
//
//
//!!! The nominal motor frequency, motor speed and the nominal motor current must 
//    be transferred to ensure the block functions correctly.
//
//
//Settings at DFE32B:
//
//1. Set IP address via Software: 
//
//2. Execute auto setup at DFE32B by setting DIP switch 2 (AS) to ON
//   All FCs must be switched on and the SBus address set
//   With the auto setup function (DIP switch "AS") it is possible to set up 
//   DFE32B as the gateway without a PC. The function is executed once when the 
//   DIP switch is switched on. The DIP switch must then remain on. The function 
//   can be executed again by switching the DIP switch off and on again.
//
//Frequency converter settings
//
//1. P100 Set setpoint source to SBUS -> value = 10
//
//2. P101 Set control source to SBus -> value 3
//
//3. P301 Set minimum speed in rpm (master value = 15)
//
//4. P302 Set maximum speed in rpm (factory setting = 1500)
//
//5. P303 Set current limit (in % of FC nominal current)
//   (Factory setting =150%)
//
//6. P320 Set automatic motor matching to on (standard setting)
//   (to gauge the motor at start)
//
//7. P500 Switch on speed monitoring
//   (in the case of fault messages P501 increase speed monitoring delay time)
//
//8. P601, P603 and P608 Set binary inputs to ""no function" (=0)
//   Set P602 to 1 = enable (factory setting) DI03 must be bypassed
//
//9. P604 for operation with PTC resistor set to 26 (TF message) otherwise
//   .... zeroing.
//   
//11. P881 Set SBus address of respective frequency converter (from 1 in
//    ascending order)
//
//12. P883 Bus monitoring time -> 5 [s]
//
//13. P884 Check SBus baud rate -> value 500/500 kBaud
//
//14. P870-P872 Setpoint description PA1-PA3
//       P870 = control word 1
//       P871 = speed
//       P872 = reserve
//    P873-P876 Actual value description PE1-PE3
//       P873 = status word 1
//       P874 = speed
//       P875 = output current in % of nominal current
//
AUTHOR : kal
FAMILY : AZO
NAME : standard
VERSION : 0.0
VAR_INPUT
  in_PEA_Adresse : INT ;	//Basisadresse für EA-Daten im PEA-Bereich
  in_FU_Nummer : INT ;	//FU Nummer zur Berechnung des Offsets der Peripherie-EAs
  in_Motordaten_J_N : BOOL ;	//nicht möglich => CLR
  in_Freigabe : BOOL ;	//Steuersignal 1 setzen zum Starten des FUs
  in_Linkslauf : BOOL ;	//Frequenzumformer Linkslauf ein
  in_Quittierung_Stoerung : BOOL ;	//Störung quittieren
  in_Sollfrequenz : REAL ;	//Sollfrequenz in Hz
  in_Motorleistungsfaktor : REAL ;	//nicht vorhanden => 0
  in_Motornennfrequenz : REAL ;	//Wertebereich: 0 - 100 Hz
  in_Motornenndrehzahl : REAL ;	//Wertebereich: 0 - 10000 U/min
  in_Motornennstrom : REAL ;	//Wertebereich: 0- ... A
  in_Motornennspannung : REAL ;	//nicht vorhanden => 0
  in_Motornennleistung : REAL ;	//nicht vorhanden => 0
END_VAR
VAR_OUTPUT
  out_Istfrequenz : REAL ;	//Istfrequenz in Hz
  out_Istdrehzahl : REAL ;	//Istdrehzahl in U/min
  out_Leistung : REAL ;	//nicht vorhanden => 0
  out_Drehmoment : REAL ;	//nicht vorhanden => 0
  out_Motorspannung : REAL ;	//nicht vorhanden => 0
  out_Ausgangsstrom : REAL ;	//Ausgangsstrom des FU
  out_Stoerung : BOOL ;	//1=Gerätestörung
  out_Warnung : BOOL ;
  out_Sollwert_erreicht : BOOL ;	//zeigt 1 an, wenn Istwert gleich Sollwert ist
  out_laeuft : BOOL ;	//=1 wenn Istdrehzahl > 0
  out_FB_Fehlermeldung : INT ;	//0 = ok ; sonst Fehler_Code_L2Dp
  out_Stoerungsnummer : DINT ;	//Stoerungsnummer, bzw. Betriebszustand wenn keine Störung aktiv
END_VAR
VAR
  reserve : ARRAY  [58 .. 99 ] OF BYTE ;
  Prozessdatenkanal_in : STRUCT 	//Prozesseingangsdaten
   PI1_Statuswort : STRUCT
    Zustand_Fehlercode : BYTE ;
    Endstufe_freigegeben : BOOL ;
    Umrichter_betriebsbereit : BOOL ;
    PA_Daten_freigegeben : BOOL ;
    reserve_3 : BOOL ;
    reserve_4 : BOOL ;
    Stoerung_Warnung : BOOL ;
    reserve_6 : BOOL ;	//0 = 1. Satz; 1 = 2. Satz
    reserve_7 : BOOL ;	//0 = 1. Satz; 1 = 2. Satz
   END_STRUCT ;
   PI2_Istdrehzahl : INT ;
   PI3_Ausgangsstrom : INT ;
  END_STRUCT ;
  Prozessdatenkanal_out : STRUCT 	//Prozessausgangsdaten
   PO1_Steuerwort : STRUCT
    Drehrichtung : BOOL ;	//0 = rechts; 1 = links
    Motorpoti_auf : BOOL ;	//00=11= keine Änderung; 01=Hochlauf, 02=Tieflauf
    Motorpoti_ab : BOOL ;
    Festsollwerte_0 : BOOL ;	//00 = Feldbus
    Festsollwerte_1 : BOOL ;
    Festsollwert_Umschaltung : BOOL ;
    reserve_14 : BOOL ;
    reserve_15 : BOOL ;
    Reglersperre : BOOL ;	//Freigabe = '110', sonst Halt
    Freigabe_Schnellstop : BOOL ;
    Freigabe_Normalhalt : BOOL ;
    reserve_3 : BOOL ;
    reserve_4 : BOOL ;
    reserve_5 : BOOL ;	//0 = 1.Satz; 1 = 2.Satz
    Reset_Stoerung : BOOL ;	//0 = 1.Satz; 1 = 2.Satz
    reserve_7 : BOOL ;
   END_STRUCT ;
   PO2_Solldrehzahl : INT ;	//in %
   PO3_keine_Fkt : INT ;
  END_STRUCT ;
  Datenuebertragung : STRUCT
   Schritt_aktiv : BOOL ;
  END_STRUCT ;
  reserve_1 : ARRAY  [122 .. 137 ] OF BYTE ;
END_VAR
VAR_TEMP
  IO_Adr_Parameterkanal : WORD ;
  IO_Adr_Prozessdatenkanal : WORD ;
  Ret_Val_SFC14_1 : INT ;
  Ret_Val_SFC14_2 : INT ;
  Ret_Val_SFC15_1 : INT ;
  Ret_Val_SFC15_2 : INT ;
  SimFactor : REAL ;	//(001)
  Solldrehzahl_tmp : REAL ;
END_VAR
BEGIN
NETWORK
TITLE = Bausteinende wenn PEA-Adresse = 0
      L     #in_PEA_Adresse;
      L     0;
      ==I;
      BEC;
NETWORK
TITLE = Simulation
//Über die Simulaitonsmerker "M 0.5 Simulation intern" oder "M 0.6 Simulation 
//AVP" 
//wird die Funktion des FUs simuliert:
//- Fehler werden zurückgesetzt
//- Bei Freigabe Istdrehzahl=Solldrehzahl, Betrieb und Solldrehzahl erreicht = 
//True
//(002) Überarbeitung 
      O     M 0.5;
      O     M 0.6;
      JCN   NSIM;
// <<(002)
      SET;
      R     #out_Stoerung;
      R     #out_Warnung;
// >>(002)
      L     L#0;
      T     #out_Stoerungsnummer;
      A     #in_Freigabe;
      =     #out_laeuft;
      =     #out_Sollwert_erreicht;
      L     #in_Sollfrequenz;
      JC    SIMD;
      L     0.000000e+00;
SIMD: T     #out_Istfrequenz;
// <<(002)
// Faktor berechnen
//     L     #out_Istfrequenz
//     L     #in_Motornennfrequenz
//      /R    
//     T     #SimFactor
// Istdrehzahl
//     L     #in_Motornenndrehzahl
//     L     #SimFactor
//      *R    
//     T     #out_Istdrehzahl
// Istleistung
//     L     #in_Motornennleistung
//     L     #SimFactor
//      *R    
//     T     #out_Leistung
// Istspannung
//     L     #in_Motornennspannung
//     L     #SimFactor
//      *R    
//     T     #out_Motorspannung
// Iststrom
//     L     #in_Motornennstrom
//     L     #SimFactor
//      *R    
//     T     #out_Ausgangsstrom
// >>(002)
      BEU;
NSIM: NOP   0;
NETWORK
TITLE = Daten von FU einlesen
//FU-Daten auslesen mit SFC14
//PEA_Adresse zeigt auf den Anfang des EA-Bereiches.
// 6-Byte Prozessdatenkanal
// <<(002)
      L     #in_FU_Nummer;
      +     -1;
      L     6;	// Länge eines Parameterkanals je FU
      *I;
      L     #in_PEA_Adresse;
      +I;
      T     #IO_Adr_Prozessdatenkanal;	// Daten des jeweiligen FU = PEA-Adresse + 8 Byte + (FU-Nr. - 1) * 6
// >>(002)
      CALL  SFC 14 (
           LADDR                    := #IO_Adr_Prozessdatenkanal,
           RET_VAL                  := #Ret_Val_SFC14_2,
           RECORD                   := #Prozessdatenkanal_in);
NETWORK
TITLE = Istdrehzahl auswerten
//Istdrehzahl in 0,2 U/min
      L     #Prozessdatenkanal_in.PI2_Istdrehzahl;
      ITD;
      DTR;
      L     5.000000e+00;
      /R;
      T     #out_Istdrehzahl;
NETWORK
TITLE = Istfrequenz auswerten
//Istfrequenz (in Hz) = Istdrehzahl (in 0,2 U/min) / 5 * Nennfrequenz / 
//Nenndrehzahl 
      L     #out_Istdrehzahl;
      L     #in_Motornennfrequenz;
      *R;
      L     #in_Motornenndrehzahl;
      /R;
      T     #out_Istfrequenz;	// in Hz
      L     0.000000e+00;	//  wenn kleiner 0 dann negieren 
      <R;
      JCN   E_IF;
      L     #out_Istfrequenz;
      L     -1.000000e+00;
      *R;
      T     #out_Istfrequenz;
E_IF: NOP   0;
NETWORK
TITLE = Stromwert auswerten
      L     #Prozessdatenkanal_in.PI3_Ausgangsstrom;	// in % des FU-Nennstomes 
      ITD;
      DTR;
      L     1.000000e+03;
      /R;
      L     #in_Motornennstrom;
      *R;
      T     #out_Ausgangsstrom;
NETWORK
TITLE = Betriebsmeldung
      A(;
      L     #out_Istfrequenz;
      L     1.000000e+00;
      >R;
      );
      =     #out_laeuft;
NETWORK
TITLE = Sollwert erreicht
      L     #in_Sollfrequenz;
      L     #out_Istfrequenz;
      -R;
      ABS;
      L     1.000000e+00;
      <R;
      =     #out_Sollwert_erreicht;
NETWORK
TITLE = Störungsbit auswerten
//Störungsbit aus Statuswort auswerten
      AN    #Prozessdatenkanal_in.PI1_Statuswort.Umrichter_betriebsbereit;
      A     #Prozessdatenkanal_in.PI1_Statuswort.Stoerung_Warnung;
      O(;
      L     #out_FB_Fehlermeldung;
      L     0;
      <>I;
      );
      O(;
      L     #out_Stoerungsnummer;
      L     0;
      <>D;
      );
      =     #out_Stoerung;
NETWORK
TITLE = Störung resetten
//Störung resetten
//NW Warnungsbit Verschoben (002)
      A     #in_Quittierung_Stoerung;
      A     #Prozessdatenkanal_in.PI1_Statuswort.Stoerung_Warnung;
      =     #Prozessdatenkanal_out.PO1_Steuerwort.Reset_Stoerung;
NETWORK
TITLE = Gerätezustand / Störungsnummer des Frequenzumformers auslesen
//Gerätezustand wenn Bit Störung/Warnung = 0
//Störungsnummer wenn Bit Störung/Warnung = 1
      L     #Prozessdatenkanal_in.PI1_Statuswort.Zustand_Fehlercode;
      ITD;
      T     #out_Stoerungsnummer;
// Störmeldung nur wenn Bit Störung = 1
      A     #Prozessdatenkanal_in.PI1_Statuswort.Stoerung_Warnung;
      JC    ESTO;
      L     0;
      T     #out_Stoerungsnummer;
ESTO: NOP   0;
NETWORK
TITLE = Freigabebefehl bearbeiten
      CLR;
      =     #Prozessdatenkanal_out.PO1_Steuerwort.Reglersperre;
      SET;
      =     #Prozessdatenkanal_out.PO1_Steuerwort.Freigabe_Schnellstop;
      A     #in_Freigabe;
      =     #Prozessdatenkanal_out.PO1_Steuerwort.Freigabe_Normalhalt;
NETWORK
TITLE = Belegung der restlichen Steuerbits
      CLR;
      =     #Prozessdatenkanal_out.PO1_Steuerwort.reserve_3;
      =     #Prozessdatenkanal_out.PO1_Steuerwort.reserve_4;
      =     #Prozessdatenkanal_out.PO1_Steuerwort.reserve_5;
      =     #Prozessdatenkanal_out.PO1_Steuerwort.reserve_7;
      =     #Prozessdatenkanal_out.PO1_Steuerwort.Motorpoti_auf;
      =     #Prozessdatenkanal_out.PO1_Steuerwort.Motorpoti_ab;
      =     #Prozessdatenkanal_out.PO1_Steuerwort.Festsollwerte_0;
      =     #Prozessdatenkanal_out.PO1_Steuerwort.Festsollwerte_1;
      =     #Prozessdatenkanal_out.PO1_Steuerwort.Festsollwert_Umschaltung;
      =     #Prozessdatenkanal_out.PO1_Steuerwort.reserve_14;
      =     #Prozessdatenkanal_out.PO1_Steuerwort.reserve_15;
NETWORK
TITLE = Solldrehzahl
//Solldrehzahl (in 0,2 HZ) 
//Sollfrequenz (in Hz) * 5 * Nenndrehzahl / Nennfrequenz
//(002) Begrenzung Solldrehzahl auf INT 
//
      L     #in_Sollfrequenz;
      L     #in_Motornenndrehzahl;
      *R;
      L     5.000000e+00;
      *R;
      L     #in_Motornennfrequenz;
      /R;
      T     #Solldrehzahl_tmp;	//(002)
      L     3.276700e+04;	//(002)
      >R;	//(002)
      JCN   SD_1;	//(002)
// maximale Drehzahl ausgeben wenn angeforderte größer als Maximalwert ist
      L     3.276700e+04;	//(002)
      RND;	//(002)
      T     #Prozessdatenkanal_out.PO2_Solldrehzahl;	//(002)
      JU    SD_L;	//(002)
// Drehzahl ausgeben wenn angeforderte kleiner als Maximalwert ist
SD_1: L     #Solldrehzahl_tmp;	//(002)
      RND;	//(002)
      T     #Prozessdatenkanal_out.PO2_Solldrehzahl;	//(002)
SD_L: AN    #in_Linkslauf;	//(002)
      JC    E_SD;	//(002)
      L     #Prozessdatenkanal_out.PO2_Solldrehzahl;
      L     -1;
      *I;
      T     #Prozessdatenkanal_out.PO2_Solldrehzahl;
E_SD: NOP   0;
NETWORK
TITLE = Warnungsbit
// (002) Verschoben + Änderung
      A     #Prozessdatenkanal_in.PI1_Statuswort.Umrichter_betriebsbereit;
      A     #Prozessdatenkanal_in.PI1_Statuswort.Stoerung_Warnung;
      O(;	//(002)
      L     #Solldrehzahl_tmp;	//(002)
      L     3.276700e+04;	//(002)
      >=R;	//(002)
      );	//(002)
      O(;	//(002)
      L     #Solldrehzahl_tmp;	//(002)
      L     -3.276700e+04;	//(002)
      <=R;	//(002)
      );	//(002)
      =     #out_Warnung;
NETWORK
TITLE = Netzwerk für nicht unterstützte Funktionen
//Zur Standardisierung der E/A-Parameter aller FUs
      L     0.000000e+00;
      T     #out_Leistung;
      T     #out_Drehmoment;
      T     #out_Motorspannung;
NETWORK
TITLE = Daten an FU senden
// 6-Byte Prozessdatenkanal
      CALL  SFC 15 (
           LADDR                    := #IO_Adr_Prozessdatenkanal,
           RECORD                   := #Prozessdatenkanal_out,
           RET_VAL                  := #Ret_Val_SFC15_2);
NETWORK
TITLE = Fehlercode L2Dp in FB_Fehlermeldung
      L     0;
      L     #Ret_Val_SFC14_2;
      <>I;
      JC    Fehl;
      L     0;
      L     #Ret_Val_SFC15_2;
      <>I;
      JC    Fehl;
      L     0;
Fehl: T     #out_FB_Fehlermeldung;
END_FUNCTION_BLOCK

FUNCTION FC 2 : VOID
TITLE = Taktgeber
//Erstellung:
//Datum        Bearbeiter                                                 Version
//--------------------------------------------------------------------------------
//16.12.97     R.Schaffert (sra)                                          01.00.00
//  
//Änderungen:
//Nr. Datum    Bearb Änderung                                       Marke  Version
//--------------------------------------------------------------------------------
//01  09.03.99 sra   Variabler Takteingang                          ()    01.01.00
//02  18.03.99 sra   Fehlerbeseitigung                              ()    01.01.01
//03  01.04.99 jm    Taktzähler auch bei Dauertakt aktiv            ()    01.01.02
//04  14.04.99 sra   Fehlerbeseitigung                              ()    01.01.03
//05  20.12.00 sra   Taktanz.err. rücksetzen bei Dauertakt          ()    01.01.04
//
//________________________________________________________________________________
//Beschreibung:
//
//Diese Funktion generiert ein beliebiges Taktsignal ohne Verwendung eines Timers.
//Es muß ein Impulssignal der Standardimpulse MB4 angelegt werden das über die 
//Taktmerker der CPU und dem Standardbaustein FC13 generiert wird
//Die Zykluszeit muß dabei kleiner sein als das verwendete Taktsignal / 2
//
//Achtung !
//- Am Parameter "in_Rueckmeldung" darf nicht "true" oder "false" angelegt 
//  werden, sondern es muss dem Ausgangssignal "io_Taktausgang" folgen ! 
//- Bei Angabe von z.B. "in_Sollanzahl_Takte" = 5 wird der Parameter 
//  "io_Taktzaehler" von 0..4 hochgezählt
//
AUTHOR : sra
FAMILY : Takt
NAME : Takt_TN
VERSION : 0.0
VAR_INPUT
  in_Freigabe : BOOL ;	//Freigabe Takt
  in_Rueckmeldung : BOOL ;	//Rueckmeldung z.B. Eingang ein
  in_Start_mit_Impuls : BOOL ;	//Takt mit positivem Impuls starten
  in_Dauertakt : BOOL ;	//Dauertakt ? (1=Ja / 0=Nein)
  in_Impuls : BOOL ;	//Impulseingang Takt
  in_Impulszeit_in_100ms : INT ;	//Impulszeit in 100ms
  in_Impulszeit : REAL ;	//Impulszeit fuer Takt in Sekunden
  in_Pausezeit : REAL ;	//Pausezeit fuer Takt in Sekunden
  in_Sollanzahl_Takte : INT ;	//Sollanzahl Takte wenn nicht Dauertakt
END_VAR
VAR_IN_OUT
  io_Taktausgang : BOOL ;	//Taktausgang
  io_Taktanzahl_erreicht : BOOL ;	//Meldung Taktanzahl erreicht
  io_Zeitzaehler : REAL ;	//Zeitzähler (abgelaufene Zeit)
  io_Taktzaehler : INT ;	//Taktzähler
END_VAR
BEGIN
NETWORK
TITLE = Rücksetzen der Zähler und Merker
//Wenn keine Freigabe mehr anliegt werden die in_out Parameter auf 0 gesetzt.
//
      A     #in_Freigabe;
      JC    Strt;
      L     1.000000e-02;
      T     #io_Zeitzaehler;
      L     0;
      T     #io_Taktzaehler;
      SET;
      R     #io_Taktausgang;
      R     #io_Taktanzahl_erreicht;
      BEU;
NETWORK
TITLE = Dauerimpuls oder Dauerpause
Strt: NOP   0;
      L     #in_Impulszeit;
      L     0.000000e+00;
      ==R;
      R     #io_Taktausgang;
      BEC;
      L     #in_Pausezeit;
      L     0.000000e+00;
      ==R;
      S     #io_Taktausgang;
      BEC;
NETWORK
TITLE = Start Takt mit Impuls
//Wenn der Takt mit einem Impuls gestartet werden soll, wird der Ausgang beim 
//Start des Taktes zunächst auf 1 gesetzt.
//Bedingung: Zeitzähler und Taktzähler müssen 0 sein
      A     #in_Freigabe;
      A     #in_Start_mit_Impuls;
      A(;
      A(;
      L     #io_Zeitzaehler;
      L     1.000000e-02;
      ==R;
      );
      A(;
      L     #io_Taktzaehler;
      L     0;
      ==I;
      );
      O;
      A     #in_Dauertakt;
      A     #io_Taktanzahl_erreicht;
      );
      S     #io_Taktausgang;
NETWORK
TITLE = Taktanzahl erreicht ?
//Abfrage ob Taktanzahl erreicht ist
      L     #io_Taktzaehler;
      L     #in_Sollanzahl_Takte;
      >=I;
      S     #io_Taktanzahl_erreicht;
      A     #in_Dauertakt;
      A     #io_Taktanzahl_erreicht;
      JCN   NCCR;	//No Clock Counter Reset
      L     0;
      T     #io_Taktzaehler;
      SET;
      R     #io_Taktanzahl_erreicht;
NCCR: NOP   0;	//No Clock Counter Reset
NETWORK
TITLE = Impuls-Phase des Taktes
//Erhöhung des Zeitzählers während der Impulsphase
//Ist die Sollzeit erreicht wird der Taktzähler erhöht, der Taktausgang 
//zurückgesetzt und der Zeitzähler wieder auf 0 gesetzt
      AN    #io_Taktausgang;
      JC    P_PH;	// wenn Taktausgang nicht gesetzt ist -> Pausephase 
      A     #in_Rueckmeldung;	// solange keine Rückmeldung -> Zeit läuft nicht
      JC    RM_I;
      L     0.000000e+00;
      T     #io_Zeitzaehler;	// Zeitzähler löschen wenn keine Rückmeldung
      JU    ENDE;
RM_I: NOP   0;
      AN    #in_Impuls;
      JC    IMP0;
      L     #in_Impulszeit_in_100ms;
      ITD;
      DTR;
      L     1.000000e-01;
      *R;
      L     #io_Zeitzaehler;	// Zeitzähler erhöhen
      +R;
      T     #io_Zeitzaehler;
      L     #in_Impulszeit;
      <R;
      JC    IMP0;
      SET;
      R     #io_Taktausgang;
      L     #io_Taktzaehler;
      INC   1;
      T     #io_Taktzaehler;
      L     0.000000e+00;
      T     #io_Zeitzaehler;	// Zeitzähler löschen
IMP0: NOP   0;
NETWORK
TITLE = Pause-Phase des Taktes
//Erhöhung des Zeitzählers während der Pausephase
//Ist die Sollzeit erreicht wird der Taktzähler erhöht, der Taktausgang 
//gesetzt und der Zeitzähler wieder auf 0 gesetzt.
//Ist die Solltaktzahl erreicht erfolgt keine weiter Bearbeitung des Netzwerks
P_PH: O     #io_Taktausgang;
      O     #io_Taktanzahl_erreicht;
      JC    ENDE;	// wenn Taktausgang gesetzt ist -> ENDE
      AN    #in_Rueckmeldung;	// solange Rückmeldung -> Zeit läuft nicht
      JC    RM_P;
      L     0.000000e+00;
      T     #io_Zeitzaehler;	// Zeitzähler löschen wenn keine Rückmeldung
      JU    ENDE;
RM_P: NOP   0;
      AN    #in_Impuls;
      JC    ENDE;
      L     #in_Impulszeit_in_100ms;
      ITD;
      DTR;
      L     1.000000e-01;
      *R;
      L     #io_Zeitzaehler;	// Zeitzähler erhöhen
      +R;
      T     #io_Zeitzaehler;
      L     #in_Pausezeit;
      <R;
      JC    ENDE;
      SET;
      S     #io_Taktausgang;
      L     0.000000e+00;
      T     #io_Zeitzaehler;	// Zeitzähler löschen
ENDE: NOP   0;
END_FUNCTION

FUNCTION FC 3 : VOID
TITLE = Ein- / Ausschaltverzögerung
//Erstellung:
//Datum        Bearbeiter                                                 Version
//--------------------------------------------------------------------------------
//27.05.97     R.Schaffert (sra)                                          01.00.00
//  
//Änderungen:
//Nr. Datum    Bearb Änderung                                       Marke  Version
//--------------------------------------------------------------------------------
//01  05.02.1999  hus      Parameter "Reset" eingeführt             ()    01.01.00
//02  22.03.1999  sra      Fehlerbeseitigung                        ()    01.01.01
//03  25.08.1999  jm       SV inkl. Reset (getestet)                ()    01.02.00
//04  27.09.1999  jm       SI inkl. Reset (getestet)                ()    01.03.00
//05  26.05.2002  jm       SZ inkl. Reset (getestet): Zeitzähler    ()    01.04.00
//06  22.05.2007  sra      Zeitzaehler läuft bei SE weiter          (006) 01.04.01
//
//________________________________________________________________________________
//Beschreibung:
//
//Diese Funktion generiert eine Ein- bzw. Ausschaltverzögerung ohne Verwendung 
//eines Timers. 
//
//Es muß ein Impulssignal "in_Impuls" der Standardimpulse MB4 angelegt werden, 
//das durch die Angabe der Taktzeit in 1/100ms "in_Impulszeit_in_100ms" 
//spezifiziert wird.
//
//Wird der Eingang "Reset" gesetzt, wird der Ausgang zurückgesetzt und der 
//Zeitzähler wird auf 0 gesetzt.
//
//SE: Durch Auswahl von "E" als Verzögerungsart wird eine Einschaltverzögerung 
//gestartet sobald "in_Freigabe" vorhanden ist. Der Ausgang "io_Ausgangssignal" 
//wird nach Ablauf der Verzögerungszeit "in_Verzoegerungszeit" auf 1 gesetzt und 
//steht dann solange an bis die Freigabe nicht mehr vorhanden ist. Der Eingang 
//"in_Reset"  bewirkt eine Nullung der Istzeit und ein Rücksetzen des Ausgangs. 
//Wird der Eingang "in_Reset" weggenommen so startet die Verzögerungszeit von 
//vorne, es sei denn "in_Freigabe" ist dann nicht mehr vorhanden.
//
//SA: Durch Auswahl von "A" als Verzögerungsart wird eine Ausschaltverzögerung 
//gestartet sobald "in_Freigabe" vorhanden ist. Der Ausgang wird sofort mit 
//dem Signal "in_Freigabe" auf 1 gesetzt. Sobald die Freigabe nicht mehr 
//vorhanden ist wird die Ausschaltverzögerung gestartet. Der Ausgang 
//"io_Ausgangssignal" steht weiterhin auf 1. Nach Ablauf der Verzögerungszeit 
//"in_Verzoegerungszeit" wird der Ausgang "io_Ausgangssignal" auf 0 gesetzt. Der 
//Eingang "in_Reset" bewirkt eine Nullung der Istzeit und ein Rücksetzen des 
//Ausgangs. Wird der Eingang "in_Reset" weggenommen so startet die Funktion von 
//vorne, es sei denn "in_Freigabe" ist dann nicht mehr vorhanden.
//
//SV: Durch Auswahl von "V" als Verzögerungsart wird ein verlängerter Impuls 
//gestartet sobald "in_Freigabe" vorhanden ist. Der Ausgang "io_Ausgangssignal" 
//wird für die Verzögerungszeit "in_Verzoegerungszeit" auf 1 gesetzt, unabhängig 
//vom Eingang "in_Freigabe". Der Eingang "in_Reset" bewirkt eine Nullung der 
//Istzeit und ein Rücksetzen des Ausgangs. Wird der Eingang "in_Reset" 
//weggenommen so startet der Impuls von vorne, es sei denn "in_Freigabe" ist dann 
//nicht mehr vorhanden.  
//
//SI: Durch Auswahl von "I" als Verzögerungsart wird ein Impuls gestartet sobald 
//"in_Freigabe" vorhanden ist. Der Ausgang "io_Ausgangssignal" wird für die 
//bestimmte Zeit auf 1 gesetzt, abhängig vom Eingang "in_Freigabe". Der Eingang 
//"Reset" bewirkt eine Nullung der Istzeit und ein Rücksetzen des Ausgangs 
//"io_Ausgangssignal". Wird der Eingang "Reset" weggenommen so startet der Impuls 
//von vorne, es sei denn "in_Freigabe" ist dann nicht mehr vorhanden.
//
//SZ: Diese Funktion kann als Zeitzähler bezeichnet werden. Sobald "in_Freigabe" 
//vorhanden ist wird die Zeit hochgezählt. Ohne "in_Freigabe" bleibt die Zeit 
//stehen, sobald "in_Freigabe" wieder vorhanden ist wird weiter gezählt. Ist die 
//Sollzeit "in_Verzoegerungszeit" erreicht und "in_Freigabe" geht weg, wird der 
//Zeitzähler rückgesetzt. Der Eingang "Reset" bewirkt eine Nullung der Istzeit 
//und ein Rücksetzen des Ausgangs "io_Ausgangssignal". Wird der Eingang "Reset" 
//weggenommen so startet der Zeitzähler von vorne, es sei denn "in_Freigabe" ist 
//dann nicht mehr vorhanden.
AUTHOR : hus
FAMILY : AZO
VERSION : 0.1
VAR_INPUT
  in_Freigabe : BOOL ;	//Freigabe Timernachbildung
  in_Reset : BOOL ;	//Reset (z.B. Steuerspannung aus)
  in_Impuls : BOOL ;	//Impulseingang (M1.7)
  in_Impulszeit_in_100ms : INT ;	//Impulszeit in 100ms (MW6)
  in_Verzoegerungsart : CHAR ;	//'E'=Einschalt-,'A'=Ausschaltverz.,'V'=verl.Impuls,'I'= Impuls,'Z'=Zeitzähler
  in_Verzoegerungszeit : REAL ;	//Verzögerungszeit in Sekunden
END_VAR
VAR_IN_OUT
  io_Ausgangssignal : BOOL ;	//Timerausgang
  io_Zeitzaehler : REAL ;	//Zeitzähler (abgelaufene Zeit)
END_VAR
BEGIN
NETWORK
TITLE = Einschaltverzögerung
//Einschaltverzögerung
      L     #in_Verzoegerungsart;
      L     'E';
      <>I;
      JC    E1;
      A     #in_Freigabe;
      JC    SE;
      SET;
      R     #io_Ausgangssignal;
      L     0.000000e+00;
      T     #io_Zeitzaehler;
      JU    E1;
//    O     #io_Ausgangssignal // (006)
SE:   ON    #in_Impuls;
      JC    E1;
      L     #in_Impulszeit_in_100ms;
      ITD;
      DTR;
      L     1.000000e-01;
      *R;
      L     #io_Zeitzaehler;
      +R;
      T     #io_Zeitzaehler;
      L     #in_Verzoegerungszeit;
      >=R;
      S     #io_Ausgangssignal;
E1:   NOP   0;
NETWORK
TITLE = Ausschaltverzögerung
//Ausschaltverzögerung
      L     #in_Verzoegerungsart;
      L     'A';
      <>I;
      JC    E2;
      AN    #in_Freigabe;
      JC    SA;
      SET;
      S     #io_Ausgangssignal;
      L     0.000000e+00;
      T     #io_Zeitzaehler;
      JU    E2;
SA:   ON    #io_Ausgangssignal;
      ON    #in_Impuls;
      JC    E2;
      L     #in_Impulszeit_in_100ms;
      ITD;
      DTR;
      L     1.000000e-01;
      *R;
      L     #io_Zeitzaehler;
      +R;
      T     #io_Zeitzaehler;
      L     #in_Verzoegerungszeit;
      >=R;
      R     #io_Ausgangssignal;
E2:   NOP   0;
NETWORK
TITLE = Verlängerter Impuls
//Verlängerter Impuls
      L     #in_Verzoegerungsart;
      L     'V';
      <>I;
      JC    E3;
      O     #in_Freigabe;
      O     #io_Ausgangssignal;
      JC    SV;
      CLR;
      =     #io_Ausgangssignal;
      L     0.000000e+00;
      T     #io_Zeitzaehler;
      JU    E3;
SV:   A     #in_Freigabe;
      S     #io_Ausgangssignal;
      L     #io_Zeitzaehler;
      L     #in_Verzoegerungszeit;
      >=R;
      R     #io_Ausgangssignal;
      ON    #in_Impuls;
      ON    #io_Ausgangssignal;
      JC    E3;
      L     #in_Impulszeit_in_100ms;
      ITD;
      DTR;
      L     1.000000e-01;
      *R;
      L     #io_Zeitzaehler;
      +R;
      T     #io_Zeitzaehler;
      L     #in_Verzoegerungszeit;
      >=R;
      R     #io_Ausgangssignal;
E3:   NOP   0;
NETWORK
TITLE = Impuls
//Impuls
      L     #in_Verzoegerungsart;
      L     'I';
      <>I;
      JC    E4;
      A     #in_Freigabe;
      JC    SI;
      CLR;
      =     #io_Ausgangssignal;
      L     0.000000e+00;
      T     #io_Zeitzaehler;
      JU    E4;
SI:   A     #in_Freigabe;
      S     #io_Ausgangssignal;
      L     #io_Zeitzaehler;
      L     #in_Verzoegerungszeit;
      >=R;
      R     #io_Ausgangssignal;
      ON    #in_Impuls;
      ON    #io_Ausgangssignal;
      JC    E4;
      L     #in_Impulszeit_in_100ms;
      ITD;
      DTR;
      L     1.000000e-01;
      *R;
      L     #io_Zeitzaehler;
      +R;
      T     #io_Zeitzaehler;
      L     #in_Verzoegerungszeit;
      >=R;
      R     #io_Ausgangssignal;
E4:   NOP   0;
NETWORK
TITLE = Zeitzähler 'Z'
//Einschaltverzögerung
      L     #in_Verzoegerungsart;
      L     'Z';
      <>I;
      JC    E5;
      AN    #in_Freigabe;
      A     #io_Ausgangssignal;
      JCN   SZ;	// Zeitzähler wird gelöscht, wenn Zeit abgelaufen und FRG weg geht
      SET;
      R     #io_Ausgangssignal;
      L     0.000000e+00;
      T     #io_Zeitzaehler;
      JU    E5;
SZ:   O     #io_Ausgangssignal;
      ON    #in_Freigabe;
      ON    #in_Impuls;
      JC    E5;
      L     #in_Impulszeit_in_100ms;
      ITD;
      DTR;
      L     1.000000e-01;
      *R;
      L     #io_Zeitzaehler;
      +R;
      T     #io_Zeitzaehler;
      L     #in_Verzoegerungszeit;
      >=R;
      S     #io_Ausgangssignal;
E5:   NOP   0;
NETWORK
TITLE = Rücksetzen Ausschaltverzögerung wenn Reseteingang = "True". 
      AN    #in_Reset;
      JC    E6;
      A     #io_Ausgangssignal;
      R     #io_Ausgangssignal;
      L     0.000000e+00;
      T     #io_Zeitzaehler;
E6:   NOP   0;
END_FUNCTION

FUNCTION FC 4 : VOID
TITLE = BlockTransfer mit ANY-Zeiger als Quelle
//Erstellung:
//Datum        Bearbeiter                                                Version
//--------------------------------------------------------------------------------
//09.03.99     R.Schaffert (sra)                                         V01.00.00
//
//Änderungen:
//Nr. Datum    Bearb Beschreibung                                   Marke Version
//--------------------------------------------------------------------------------
//01 30.06.99  sra   Fehlerbeseitigung                                    01.00.01
//02 27.01.04  gea   Fehlerbeseitigung Quell-DW > 8192              (002) 01.00.02
//03 13.12.05  sra   Fehlerbeseitigung Ziel-DW > 8192               (003) 01.00.03
//04 10.06.10  sra   Bereich > 32767 kopieren                       (004) 01.00.04
//________________________________________________________________________________
//Funktion:
//
//Blocktranferfunktion mit Systemfunktion SFC20
//-Bei "in_Ziel_Typ" = 'E' werden die Aktualwerte des in "in Quelle" definierten 
// Bereiches an den durch "in_Ziel_DW" definierten Eingangsbereich kopiert.
//-Bei "in_Ziel_Typ" = 'A' werden die Aktualwerte des in "in Quelle" definierten 
// Bereiches an den durch "in_Ziel_DW" definierten Ausgangsbereich kopiert.
//-Bei "in_Ziel_Typ" = 'M' werden die Aktualwerte des in "in Quelle" definierten 
// Bereiches an den durch "in_Ziel_DW" definierten Merkerbereich kopiert.
//-Bei "in_Ziel_Typ" = 'D' werden die Aktualwerte des in "in Quelle" definierten 
// Bereiches an den durch "in_Ziel_DB" und "in_Ziel_DW" definierten 
// Global-Datenbaustein kopiert.
//-Bei "in_Ziel_Typ" = 'I' werden die Aktualwerte des in "in Quelle" definierten 
// Bereiches an den durch "in_Ziel_DW" definierten Zielbereich des aktuellen 
// Instanz-Datenbausteines kopiert.
//
//An diesen Funktionsbaustein und den SFC20 werden Zeiger (ANY-Zeiger) angelegt, 
//die die Datenquelle definieren. Zeiger ist folgendermaßen aufgebaut:
//     Byte n       B#16#10 
//     Byte n+1     Datentyp (Bool, Byte, usw.)
//     Byte n+2     Anzahl der Datentypen die kopiert werdn sollen (2 Byte)
//     Byte n+4     Datenbausteinnummer (2 Byte)
//     Byte n+6     Bereichszeiger (4 Byte)
//
//Aufbau des bereichsübergreifenden Zeigers:  10000ZZZ 00000yyy yyyyyyyy yyyyyxxx
//      z = Operandenbereich (codiert)
//      y = Byte-Adresse
//      x = Bit-Adresse
//
AUTHOR : sra
FAMILY : AZO
VERSION : 0.0
VAR_INPUT
  in_Quelle : ANY ;	//ANY-Zeiger auf Quelle
  in_Ziel_Typ : CHAR ;	//E=Eingang, A=Ausgang, M=Merker, D=DB, I=Instanz-DB
  in_Ziel_DB : INT ;	//Ziel-DB bei DW-Transfer
  in_Ziel_DW : INT ;	//Ziel-DW Byte-Adresse des Ziels
END_VAR
VAR_OUTPUT
  out_Fehler : INT ;	//1=Ziel-Typ ungültig, 2=DB existiert nicht, 3= DB zu kurz, SFC20 Fehlermeldung
END_VAR
VAR_TEMP
  Quellzeiger : ANY ;
  Zielzeiger : ANY ;
  Quell_DB : INT ;
  Quell_DW : INT ;
  Blocklaenge : INT ;
  Datentyp : BYTE ;
  SFC20_return : INT ;
  Operandenbereich : INT ;
  DB_Test_Nr : WORD ;
  DB_Test_Fehler : INT ;
  DB_Test_Anz_Byte : WORD ;
  DB_Test_Schreib_Schutz : BOOL ;
END_VAR
BEGIN
NETWORK
TITLE = Operandenbereich Quelle codieren
//Bereichscodierung für Quelltyp durchführen
//Operandenbereich im bereichsübergreifenden Zeiger
//
//Aufbau des bereichsübergreifenden Zeigers:  10000ZZZ 00000yyy yyyyyyyy yyyyyxxx
//      z = Operandenbereich (codiert)
//      y = Byte-Adresse
//      x = Bit-Adresse
//    
      L     P##in_Quelle;
      LAR1;
      L     B [AR1,P#1.0];
      T     #Datentyp;
      L     W [AR1,P#2.0];
      T     #Blocklaenge;
      L     W [AR1,P#4.0];
      T     #Quell_DB;
      L     D [AR1,P#6.0];
      L     DW#16#FFFFFF;
      AD;
      SRD   3;	//(002)
      T     #Quell_DW;
      L     D [AR1,P#6.0];
      L     DW#16#F000000;
      AD;
      SRD   24;
      T     #Operandenbereich;
NETWORK
TITLE = Quell-Datenbaustein prüfen
//Überprüfen bei Quelltyp = D,I : Baustein existiert und ist ausreichend lang
      L     #Operandenbereich;
      L     5;	//Quelle ist Instanz-DB 
      <>I;
      JC    M004;
      L     DINO;	//Nummer akt. Instanz-DB
      T     #Quell_DB;
      T     #DB_Test_Nr;
      JU    M005;
M004: L     #Operandenbereich;
      L     4;	//Quelle ist Global-DB
      <>I;
      JC    M003;
      L     #Quell_DB;
      T     #DB_Test_Nr;
M005: CALL  SFC 24 (
           DB_NUMBER                := #DB_Test_Nr,
           RET_VAL                  := #DB_Test_Fehler,
           DB_LENGTH                := #DB_Test_Anz_Byte,
           WRITE_PROT               := #DB_Test_Schreib_Schutz);
      L     #DB_Test_Fehler;
      L     0;
      ==I;
      JC    M006;
      L     2;	//DB existiert nicht
      T     #out_Fehler;
      BEU;
M006: L     #Quell_DW;
      L     #Blocklaenge;
      +D;	// (004)
      L     #DB_Test_Anz_Byte;
      <=D;	// (004)
      JC    M003;
      L     3;	//DB nicht ausreichend lang
      T     #out_Fehler;
      BEU;
M003: NOP   0;
NETWORK
TITLE = Quellezeiger belegen
//Quelle vom Typ "ANY" erstellen
      LAR1  P##Quellzeiger;
      L     B#16#10;
      T     LB [AR1,P#0.0];	//Syntax-ID ist immer 10h bei AWL
      L     #Datentyp;
      T     LB [AR1,P#1.0];	// Datentyp 
      L     #Blocklaenge;
      T     LW [AR1,P#2.0];	// Anzahl der Bytes die kopiert werden sollen
      L     #Quell_DB;
      T     LW [AR1,P#4.0];	// Datenbaustzeinnummer
      L     #Operandenbereich;
      L     128;	// 128 addieren (Bit 31 muß 1 sein)
      +I;
      SLD   24;	// 24 Stellen nach links schieben
      L     #Quell_DW;
      SLD   3;	// Quell-DW an Byte-Adresse schieben   //(002)
      +D;	// Zeiger zusammenfügen
      T     LD [AR1,P#6.0];	// siehe Aufbau Bereichszeiger NW1
NETWORK
TITLE = Operandenbereich Ziel codieren
//Bereichscodierung für Zieltyp durchführen
//Operandenbereich im bereichsübergreifenden Zeiger
//
//Aufbau des bereichsübergreifenden Zeigers:  10000ZZZ 00000yyy yyyyyyyy yyyyyxxx
//      z = Operandenbereich (codiert)
//      y = Byte-Adresse
//      x = Bit-Adresse
//    
      L     #in_Ziel_Typ;
      L     'E';	// Ziel = Eingänge
      ==I;
      L     1;
      JC    M002;
      L     #in_Ziel_Typ;
      L     'A';	// Ziel = Ausgänge
      ==I;
      L     2;
      JC    M002;
      L     #in_Ziel_Typ;
      L     'M';	// Ziel = Merker
      ==I;
      L     3;
      JC    M002;
      L     #in_Ziel_Typ;
      L     'D';	// Ziel = DB (Globaldaten)
      ==I;
      L     4;
      JC    M002;
      L     #in_Ziel_Typ;
      L     'I';	// Ziel = Instanz-DB
      ==I;
      L     5;
      JC    M002;
      L     #in_Ziel_Typ;
      L     'L';	// Ziel = Temporäre-Lokal-Daten
      ==I;
      L     6;
      JC    M002;
      L     #in_Ziel_Typ;
      L     'V';	// Ziel = temp. Lokaldaten des Vorgängerbausteins
      ==I;
      L     7;
      JC    M002;
      L     1;	// Kein gültiger Parameter -> Fehler und Ende
      T     #out_Fehler;
      BEU;
M002: T     #Operandenbereich;
NETWORK
TITLE = Ziel-Datenbaustein prüfen
//Überprüfen bei Zieltyp = D,I : Baustein existiert und ist ausreichend lang
      L     #Operandenbereich;
      L     5;	//Ziel ist Instanz-DB 
      <>I;
      JC    M007;
      L     DINO;	//Nummer akt. Instanz-DB
      T     #in_Ziel_DB;
      T     #DB_Test_Nr;
      JU    M008;
M007: L     #Operandenbereich;
      L     4;	//Ziel ist Global-DB
      <>I;
      JC    M010;
      L     #in_Ziel_DB;
      T     #DB_Test_Nr;
M008: CALL  SFC 24 (
           DB_NUMBER                := #DB_Test_Nr,
           RET_VAL                  := #DB_Test_Fehler,
           DB_LENGTH                := #DB_Test_Anz_Byte,
           WRITE_PROT               := #DB_Test_Schreib_Schutz);
      L     #DB_Test_Fehler;
      L     0;
      ==I;
      JC    M009;
      L     2;	//DB existiert nicht
      T     #out_Fehler;
      BEU;
M009: L     #in_Ziel_DW;
      L     #Blocklaenge;
      +D;	// (004)
      L     #DB_Test_Anz_Byte;
      <=D;	// (004)
      JC    M010;
      L     3;	//DB nicht ausreichend lang
      T     #out_Fehler;
      BEU;
M010: NOP   0;
NETWORK
TITLE = Zielzeiger belegen
//Ziel vom Typ "ANY" erstellen
      LAR1  P##Zielzeiger;
      L     B#16#10;
      T     LB [AR1,P#0.0];	//Syntax-ID ist immer 10h bei AWL
      L     #Datentyp;
      T     LB [AR1,P#1.0];	// Datentyp 
      L     #Blocklaenge;
      T     LW [AR1,P#2.0];	// Anzahl der Bytes die kopiert werden sollen
      L     #in_Ziel_DB;
      T     LW [AR1,P#4.0];	// Datenbaustzeinnummer
      L     #Operandenbereich;
      L     128;	// 128 addieren (Bit 31 muß 1 sein)
      +I;
      SLD   24;	// 24 Stellen nach links schieben
      L     #in_Ziel_DW;
      SLD   3;	// Quell-DW an Byte-Adresse schieben (003)
      +D;	// Zeiger zusammenfügen
      T     LD [AR1,P#6.0];	// siehe Aufbau Bereichszeiger NW1
NETWORK
TITLE = Blocktransfer
//Blocktransfer mit Systemfunktion SFC20
      CALL  SFC 20 (
           SRCBLK                   := #Quellzeiger,
           RET_VAL                  := #SFC20_return,
           DSTBLK                   := #Zielzeiger);
NETWORK
TITLE = Rückgabewert SFC20
//Rückgabewert des SFC20 übergeben
      L     #SFC20_return;
      T     #out_Fehler;
END_FUNCTION

FUNCTION FC 5 : VOID
TITLE = BlockTransfer
//Erstellung:
//Datum        Bearbeiter                                                 Version
//--------------------------------------------------------------------------------
//26.06.97     G.Herkert (hkt)                                            01.00.00
//
//Änderungen:
//Nr. Datum    Bearb Beschreibung                                   Marke Version
//--------------------------------------------------------------------------------
//01  20.05.98 sra   komplette Überarbeitung                              02.00.00
//02  29.10.98 gea   Überprüfung Länge und Existenz DBs                   02.01.00
//03  24.11.98 gea   'I' kopiert in/von akt Instanz-DB                    02.02.00
//04  10.05.99 sra   Bereichszeigerberechnung korrigiert                  02.02.01
//05  10.12.01 gea   'K' löscht Bereich                             (005) 02.03.00
//06  07.06.10 sra   Bereich > 32767 kopieren                       (006) 02.03.01
//
//________________________________________________________________________________
//Funktion:
//
//Blocktranferfunktion mit Systemfunktion SFC20
//-Bei "Quell_Typ" = 'E' werden die Aktualwerte der in "Quell_DW" definierten 
// Eingangsadressen ausgelesen und kopiert.
//-Bei "Quell_Typ" = 'A' werden die Aktualwerte der in "Quell_DW" definierten 
// Ausgangsadressen ausgelesen und kopiert.
//-Bei "Quell_Typ" = 'M' werden die Aktualwerte der in "Quell_DW" definierten 
// Merkeradressen ausgelesen und kopiert.
//-Bei "Quell_Typ" = 'D' werden die Aktualwerte der in "Quell-DB" und "Quell_DW"  
// definierten Datenworte ausgelesen und kopiert.
//-Bei "Quell_Typ" = 'I' werden die Aktualwerte der in "Quell_DW" definierten 
// Datenworte des aktuellen Instanz-DBs ausgelesen und kopiert.
//
//-Bei "Ziel_Typ" = 'E' werden die definierten Quelldaten an den durch 
// "in_Ziel_DW" definierten Eingangsbereich kopiert.
//-Bei "Ziel_Typ" = 'A' werden die definierten Quelldaten an den durch 
// "in_Ziel_DW" definierten Ausgangsbereich kopiert.
//-Bei "Ziel_Typ" = 'M' werden die definierten Quelldaten an den durch 
// "in_Ziel_DW" definierten Merkerbereich kopiert.
//-Bei "Ziel_Typ" = 'D' werden die definierten Quelldaten an den durch  
//"in_Ziel_DB" und "in_Ziel_DW" definierten Global-Datenbaustein kopiert.
//-Bei "Ziel_Typ" = 'I' werden die definierten Quelldaten an den durch  
// "in_Ziel_DW" definierten Zielbereich des aktuellen Instanz-Datenbausteines  
// kopiert.
//
//An den SFC20 werden Zeiger (ANY-Zeiger) angelegt die die Quelle und das Ziel 
//beschreiben. Zeiger sind folgendermaßen aufgebaut:
//     Byte n       B#16#10 
//     Byte n+1     Datentyp (Bool, Byte, usw.)
//     Byte n+2     Anzahl der Datentypen die kopiert werdn sollen (2 Byte)
//     Byte n+4     Datenbausteinnummer (2 Byte)
//     Byte n+6     Bereichszeiger (4 Byte)
//
//Aufbau des bereichsübergreifenden Zeigers:  10000ZZZ 00000yyy yyyyyyyy yyyyyxxx
//      z = Operandenbereich (codiert)
//      y = Byte-Adresse
//      x = Bit-Adresse
AUTHOR : hkt
FAMILY : AZO
VERSION : 0.0
VAR_INPUT
  Quell_Typ : CHAR ;	//E=Eingang, A=Ausgang, M=Merker, D=DB, I=Instanz-DB, K=Löschen
  Quell_DB : INT ;	//Quell-Datenbaustein bei DW-Transfer
  Quell_DW : INT ;	//Quell-Datenwort, Byte-Adresse der Quelle
  Ziel_Typ : CHAR ;	//E=Eingang, A=Ausgang, M=Merker, D=DB, I=Instanz-DB
  Ziel_DB : INT ;	//Ziel-Datenbaustein bei DW-Transfer
  Ziel_DW : INT ;	//Ziel-Datenwort, Byte-Adresse des Zieles
  Block_Laenge : INT ;	//Blocklänge in Byte
END_VAR
VAR_OUTPUT
  outFehler : INT ;	//1=Ziel-Typ ungültig, 2=DB existiert nicht, 3= DB zu kurz, SFC20 Fehlermeldung
END_VAR
VAR_TEMP
  Quellzeiger : ANY ;
  Zielzeiger : ANY ;
  SFC20_return : INT ;
  Operandenbereich : INT ;
  DB_Test_Nr : WORD ;
  DB_Test_Fehler : INT ;
  DB_Test_Anz_Byte : WORD ;
  DB_Test_Schreib_Schutz : BOOL ;
END_VAR
BEGIN
NETWORK
TITLE = Bereich in DB-löschen
//(005)
      A(;
      L     #Quell_Typ;
      L     'K';
      ==I;
      );
      A(;
      L     #Ziel_Typ;
      L     'D';
      ==I;
      );
      JCN   BLOE;
      CALL  FC 30 (
           DB_Nr                    := #Ziel_DB,
           DW_Anfang                := #Ziel_DW,
           Anzahl_Bytes             := #Block_Laenge,
           Wert                     := 0);
      BEU;
BLOE: NOP   0;
NETWORK
TITLE = Operandenbereich Quelle codieren
//Bereichscodierung für Quelltyp durchführen
//Operandenbereich im bereichsübergreifenden Zeiger
//
//Aufbau des bereichsübergreifenden Zeigers:  10000ZZZ 00000yyy yyyyyyyy yyyyyxxx
//      z = Operandenbereich (codiert)
//      y = Byte-Adresse
//      x = Bit-Adresse
//    
      L     #Quell_Typ;
      L     'E';	// Quelle = Eingänge
      ==I;
      L     1;
      JC    M001;
      L     #Quell_Typ;
      L     'A';	// Quelle = Ausgänge
      ==I;
      L     2;
      JC    M001;
      L     #Quell_Typ;
      L     'M';	// Quelle = Merker
      ==I;
      L     3;
      JC    M001;
      L     #Quell_Typ;
      L     'D';	// Quelle = DB (Globaldaten)
      ==I;
      L     4;
      JC    M001;
      L     #Quell_Typ;
      L     'I';	// Quelle = Instanz-DB
      ==I;
      L     5;
      JC    M001;
      L     #Quell_Typ;
      L     'L';	// Quelle = Temporäre-Lokal-Daten
      ==I;
      L     6;
      JC    M001;
      L     #Quell_Typ;
      L     'V';	// Quelle = temp. Lokaldaten des Vorgängerbausteins
      ==I;
      L     7;
      JC    M001;
      L     1;	// Kein gültiger Parameter -> Fehler und Ende
      T     #outFehler;
      BEU;
M001: T     #Operandenbereich;
NETWORK
TITLE = Quell-Datenbaustein prüfen
//Überprüfen bei Quelltyp = D,I : Baustein existiert und ist ausreichend lang
      L     #Operandenbereich;
      L     5;	//Quelle ist Instanz-DB 
      <>I;
      JC    M004;
      L     DINO;	//Nummer akt. Instanz-DB
      T     #Quell_DB;
      T     #DB_Test_Nr;
      JU    M005;
M004: L     #Operandenbereich;
      L     4;	//Quelle ist Global-DB
      <>I;
      JC    M003;
      L     #Quell_DB;
      T     #DB_Test_Nr;
M005: CALL  SFC 24 (
           DB_NUMBER                := #DB_Test_Nr,
           RET_VAL                  := #DB_Test_Fehler,
           DB_LENGTH                := #DB_Test_Anz_Byte,
           WRITE_PROT               := #DB_Test_Schreib_Schutz);
      L     #DB_Test_Fehler;
      L     0;
      ==I;
      JC    M006;
      L     2;	//DB existiert nicht
      T     #outFehler;
      BEU;
M006: L     #Quell_DW;
      L     #Block_Laenge;
      +D;	// (006)    
      L     #DB_Test_Anz_Byte;
      <=D;	// (006)    
      JC    M003;
      L     3;	//DB nicht ausreichend lang
      T     #outFehler;
      BEU;
M003: NOP   0;
NETWORK
TITLE = Quellezeiger belegen
//Quelle vom Typ "ANY" erstellen
      LAR1  P##Quellzeiger;
      L     B#16#10;
      T     LB [AR1,P#0.0];	//Syntax-ID ist immer 10h bei AWL
      L     2;
      T     LB [AR1,P#1.0];	// Datentyp = 2 (Byte)
      L     #Block_Laenge;
      T     LW [AR1,P#2.0];	// Anzahl der Bytes die kopiert werden sollen
      L     #Quell_DB;
      T     LW [AR1,P#4.0];	// Datenbaustzeinnummer
      L     #Operandenbereich;
      L     128;	// 128 addieren (Bit 31 muß 1 sein)
      +I;
      SLD   24;	// 24 Stellen nach rechts schieben
      L     #Quell_DW;
      SLD   3;	// Quell-DW an Byte-Adresse schieben 
      +D;	// Zeiger zusammenfügen
      T     LD [AR1,P#6.0];	// siehe Aufbau Bereichszeiger NW1
NETWORK
TITLE = Operandenbereich Ziel codieren
//Bereichscodierung für Zieltyp durchführen
//Operandenbereich im bereichsübergreifenden Zeiger
//
//Aufbau des bereichsübergreifenden Zeigers:  10000ZZZ 00000yyy yyyyyyyy yyyyyxxx
//      z = Operandenbereich (codiert)
//      y = Byte-Adresse
//      x = Bit-Adresse
//    
      L     #Ziel_Typ;
      L     'E';	// Ziel = Eingänge
      ==I;
      L     1;
      JC    M002;
      L     #Ziel_Typ;
      L     'A';	// Ziel = Ausgänge
      ==I;
      L     2;
      JC    M002;
      L     #Ziel_Typ;
      L     'M';	// Ziel = Merker
      ==I;
      L     3;
      JC    M002;
      L     #Ziel_Typ;
      L     'D';	// Ziel = DB (Globaldaten)
      ==I;
      L     4;
      JC    M002;
      L     #Ziel_Typ;
      L     'I';	// Ziel = Instanz-DB
      ==I;
      L     5;
      JC    M002;
      L     #Ziel_Typ;
      L     'L';	// Ziel = Temporäre-Lokal-Daten
      ==I;
      L     6;
      JC    M002;
      L     #Ziel_Typ;
      L     'V';	// Ziel = temp. Lokaldaten des Vorgängerbausteins
      ==I;
      L     7;
      JC    M002;
      L     1;	// Kein gültiger Parameter -> Fehler und Ende
      T     #outFehler;
      BEU;
M002: T     #Operandenbereich;
NETWORK
TITLE = Ziel-Datenbaustein prüfen
//Überprüfen bei Zieltyp = D,I : Baustein existiert und ist ausreichend lang
      L     #Operandenbereich;
      L     5;	//Ziel ist Instanz-DB 
      <>I;
      JC    M007;
      L     DINO;	//Nummer akt. Instanz-DB
      T     #Ziel_DB;
      T     #DB_Test_Nr;
      JU    M008;
M007: L     #Operandenbereich;
      L     4;	//Ziel ist Global-DB
      <>I;
      JC    M010;
      L     #Ziel_DB;
      T     #DB_Test_Nr;
M008: CALL  SFC 24 (
           DB_NUMBER                := #DB_Test_Nr,
           RET_VAL                  := #DB_Test_Fehler,
           DB_LENGTH                := #DB_Test_Anz_Byte,
           WRITE_PROT               := #DB_Test_Schreib_Schutz);
      L     #DB_Test_Fehler;
      L     0;
      ==I;
      JC    M009;
      L     2;	//DB existiert nicht
      T     #outFehler;
      BEU;
M009: L     #Ziel_DW;
      L     #Block_Laenge;
      +D;	// (006)    
      L     #DB_Test_Anz_Byte;
      <=D;	// (006)    
      JC    M010;
      L     3;	//DB nicht ausreichend lang
      T     #outFehler;
      BEU;
M010: NOP   0;
NETWORK
TITLE = Zielzeiger belegen
//Ziel vom Typ "ANY" erstellen
      LAR1  P##Zielzeiger;
      L     B#16#10;
      T     LB [AR1,P#0.0];	//Syntax-ID ist immer 10h bei AWL
      L     2;
      T     LB [AR1,P#1.0];	// Datentyp = 2 (Byte)
      L     #Block_Laenge;
      T     LW [AR1,P#2.0];	// Anzahl der Bytes die kopiert werden sollen
      L     #Ziel_DB;
      T     LW [AR1,P#4.0];	// Datenbaustzeinnummer
      L     #Operandenbereich;
      L     128;	// 128 addieren (Bit 31 muß 1 sein)
      +I;
      SLD   24;	// 24 Stellen nach rechts schieben
      L     #Ziel_DW;
      SLD   3;	// Quell-DW an Byte-Adresse schieben 
      +D;	// Zeiger zusammenfügen
      T     LD [AR1,P#6.0];	// siehe Aufbau Bereichszeiger NW1
NETWORK
TITLE = Blocktransfer
//Blocktransfer mit Systemfunktion SFC20
      CALL  SFC 20 (
           SRCBLK                   := #Quellzeiger,
           RET_VAL                  := #SFC20_return,
           DSTBLK                   := #Zielzeiger);
NETWORK
TITLE = Rückgabewert SFC20
//Rückgabewert des SFC20 übergeben
      L     #SFC20_return;
      T     #outFehler;
END_FUNCTION

FUNCTION FC 6 : VOID
TITLE = Datenbit_setzen oder abfragen ( Adressierung Byte )
//Erstellung:
//Datum        Bearbeiter                                                 Version
//--------------------------------------------------------------------------------
//26.06.97     H.Rüttling (rh)                                            01.00.00
//
//Änderungen:
//Nr. Datum    Bearb Beschreibung                                   Marke Version
//--------------------------------------------------------------------------------
//01  12.11.98 sra   komplette Überarbeitung                              02.00.00
//02  20.11.98 gea   Vereinfachung                                        02.00.01
//03  24.09.14 sra   Adresserweiterung (>8192)                      (003) 02.01.00
//________________________________________________________________________________
//Funktion:
//
//Die Funktion schreibt oder liest den Zustand eines Datenbits.
//Das Datenbit ist definiert durch Datenbaustein [in_DB_Nr], die 
//Anfangsbytenummer [in_Byte_Nr_Anfang] und die Bitnummer [in_Bit_Nr].
//Ist der Parameter in_Mode_Z_A = 'A' wird das Datenbit gelesen und in den 
//Parameter io_Wert geschrieben.
//Ist der Parameter in_Mode_Z_A = 'Z' wird das Datenbit entsprechende dem Zustand 
//des Parameters io_Wert geschrieben.
//
//Es können auch Bitnummern > 7 verwendet werden. Dann wird die Bytenummer 
//entsprechend dem Vielfachen von 8 erhöht.
//Z.B.: Byte 8, Bit 12 entspricht Byte 9, Bit 4
//
//!!!! in_Bit_Nr.= 0 => DBX Byte X.0 !!!!!
//!!!! in_Bit_Nr.= 1 => DBX Byte X.1 !!!!!
AUTHOR : rh
FAMILY : AZO
VERSION : 0.0
VAR_INPUT
  in_DB_Nr : INT ;	//Datenbausteinnummer
  in_Byte_Nr_Anfang : INT ;	//Byte-Nummer
  in_Bit_Nr : INT ;	//Bitnummer
  in_Mode_Z_A : CHAR ;	//Z = zuweisen; A = abfragen
END_VAR
VAR_IN_OUT
  io_Wert : BOOL ;	//Wert der gelesen/geschrieben wird
END_VAR
VAR_TEMP
  Datenbaustein : INT ;
  Byte_Adresse : INT ;
  Bit_Adresse : INT ;
END_VAR
BEGIN
NETWORK
TITLE = Datenbaustein aufschlagen
      L     #in_DB_Nr;	// Datenbaustein_NR uebergeben
      T     #Datenbaustein;
      OPN   DB [#Datenbaustein];	// Datenbaustein indiziert aufschlagen
NETWORK
TITLE = Byte Adresse berechnen
      L     #in_Bit_Nr;
      SRW   3;	// Bit_ NR durch 8 dividieren
      L     #in_Byte_Nr_Anfang;	// Ergebnis zur Wort-Adresse dazuadieren
      +D;	// (003)
      T     #Byte_Adresse;	// = Datenwort Adresse
NETWORK
TITLE = Bit_Adresse berechnen
      L     #in_Bit_Nr;
      L     W#16#7;
      AW;
      T     #Bit_Adresse;
NETWORK
TITLE = Pointer auf Datenbit berechnen
      L     #Byte_Adresse;	// DW Adresse zurecht ruecken
      SLD   3;	// DW Adresse zum Adressregister  // (003)
      L     #Bit_Adresse;	// Bit Adresse hinzufügen
      OD;	// (003)
      LAR1;	// Pointer Adresse aus Adressregister
NETWORK
TITLE = Mode Auswahl
      L     'Z';
      L     #in_Mode_Z_A;
      ==I;
      JC    ZUWE;	// Sprung Datenbit zuweisen
      L     'A';
      ==I;
      JC    ABFR;	// Sprung Datenbit abfragen
      BEU;
NETWORK
TITLE = Datenbit zuweisen 
ZUWE: A     #io_Wert;
      =     DBX [AR1,P#0.0];
      BEU;
NETWORK
TITLE = Datenbit abfragen
ABFR: A     DBX [AR1,P#0.0];
      =     #io_Wert;
END_FUNCTION

FUNCTION FC 7 : VOID
TITLE = Tabelle auslesen
//Erstellung:
//Datum        Bearbeiter                                                 Version
//--------------------------------------------------------------------------------
//30.10.98     A.Geiger (gea)                                             01.00.00
//
//Änderungen:
//Nr. Datum    Bearb Beschreibung                                   Marke Version
//--------------------------------------------------------------------------------
//01  10.05.99 sra   Bereichszeigerberechnung korrigiert                  01.00.01
//02  29.08.00 gea   Neue Konzeption(Kopieren über Schleife)              02.00.00
//03  26.10.01 gea   Fehlerbehebung DB überprüfen                   (003) 02.00.01
//04  26.10.01 gea   Fehler bei Anfangsbyte negativ                 (004) 02.00.02
//05  29.02.16 sra   Anpassung für Tabellen > 32767 Byte            (005) 02.00.03
//06  17.06.16 sra   Fehlerbeseitigung Zeigerberechnung             
//                   negative Zeilen sind ebenfalls möglich         (006) 02.00.04
//________________________________________________________________________________
//Funktion:
//
//Beschreibung: Datensatz aus Tabelle auslesen
//
//Aufbau Tabellen-DB:
//      DBB(Offset)    ... DBB(n-1)  1.Zeile
//      DBB(Offset+n)  ... DBB(2n-1) 2.Zeile
//      DBB(Offset+2n) ... DBB(3n-1) 3.Zeile
//      usw.
//
//Die Anzahl der Spalten pro Zeile (n) ist abhängig von der Länge des "Ziels".
//Das "Ziel" muß ein ANY-Zeiger auf Bytes oder eine Stuktur sein.
//Eine Überprüfung auf Existenz und Länge des Tabellen-DBs wird durchgeführt.
//
//Fehlermeldungen:
//-1 = Bereichszeiger Quelle falsch
//-2 = Bereichszeiger Ziel falsch
//-3 = Blocklänge falsch
//-4 = Datenbaustein nicht existent 
//-5 = Datenbaustein Längenfehler
//-6 = Fehler Datentyp in ANY-Zeiger
//-7 = Fehler Anfangsbyte negativ    
//
AUTHOR : gea
FAMILY : gea
VERSION : 0.0
VAR_INPUT
  in_Tabelle_DB : INT ;	//Tabellen-DB-Nr.
  in_Offset_DW : INT ;	//Offset erster Tabelleneintrag in Tabellen-DB
  in_Zeile_lesen : INT ;	//Eintrag in Tabelle, der gelesen werden soll
END_VAR
VAR_OUTPUT
  out_Fehler : INT ;	//-1=Q,-2=Z,-3=Blocklänge,-4=DB n. vorh.,-5=DB zu kurz,-6=Datentyp,-7=Anfangsbyte
END_VAR
VAR_IN_OUT
  io_Ziel : ANY ;	//Zeiger auf Zieldaten Block in den kopiert wird
END_VAR
VAR_TEMP
  G_DB_SAVE : INT ;	//Global-DB-Register
  I_DB_SAVE : INT ;	//Instanz-DB-Register
  Zeiger_Quelle : DWORD ;
  DB_Quelle : INT ;
  Zeiger_Ziel : DWORD ;
  DB_Ziel : INT ;
  Blocklaenge : INT ;
  Datentyp : BYTE ;
  Start_DBB : INT ;
END_VAR
BEGIN
NETWORK
TITLE = DB-Register sichern
      L     DBNO;
      T     #G_DB_SAVE;
      L     DINO;
      T     #I_DB_SAVE;
NETWORK
TITLE = ANY-Zeiger Ziel zerlegen
      L     P##io_Ziel;
      LAR1;
      L     B [AR1,P#1.0];
      T     #Datentyp;
      L     W [AR1,P#2.0];
      T     #Blocklaenge;
      L     W [AR1,P#4.0];
      T     #DB_Ziel;
      L     D [AR1,P#6.0];
      L     DW#16#FFFFFF;	// (006)
      AD;	// (006)
      T     #Zeiger_Ziel;
NETWORK
TITLE = Blocklänge prüfen
      L     #Blocklaenge;
      L     0;
      <=I;
      JC    BLFE;	//Blocklänge Fehler
NETWORK
TITLE = Datentyp prüfen
      L     #Datentyp;
      L     2;	//Datentyp = Byte oder Struct
      ==I;
      JCN   DTFE;
NETWORK
TITLE = Start-DBB des gewählten Eintrags
      L     #in_Zeile_lesen;
      L     1;
      -I;
      L     #Blocklaenge;
      *I;
      L     #in_Offset_DW;
      +I;
      T     #Start_DBB;	//Start des n-ten Eintrags
//      L     #Start_DBB                  //Start des n-ten Eintrags      //(004) // (006)
//      L     0                           //                                (004) // (006)
//      >=I                               //                                (004) // (006)
//      SPBN  DBBN                        //Fehler Anfangsbyte negativ    //(004) // (006)
NETWORK
TITLE = Bereichszeiger Quellzeiger
      L     W#16#84;
      CAD;
      L     #Start_DBB;
      SLD   3;
      +D;
      T     #Zeiger_Quelle;
NETWORK
TITLE = Quell-DB
      L     #in_Tabelle_DB;
      T     #DB_Quelle;
NETWORK
TITLE = DBs aufschlagen
//      L     #DB_Quelle                               //(003)
//      L     0                                        //(003)
//      <>I                                            //(003)
//      SPBN  QNDB                                     //(003)
      OPN   DB [#DB_Quelle];
      L     DBNO;
      L     0;
      <=I;
      JC    DBNX;	//Fehler DB existiert nicht
      L     #Start_DBB;
      L     #Blocklaenge;
      +D;	// (005)
      L     DBLG;
      >D;	// (005)
      JC    DBLF;	//Fehler DB Länge nicht ausreichend
      L     #DB_Ziel;
      L     0;
      <>I;
      JCN   ZNDB;
      OPN   DI [#DB_Ziel];
      L     DINO;
      L     0;
      <=I;
      JC    DBNX;	//Fehler DB existiert nicht
      L     #Zeiger_Ziel;
      SRD   3;	//Anfangsbyte (005)
      L     #Blocklaenge;
      +D;	// (005)
      L     DILG;
      >D;	// (005)
      JC    DBLF;	//Fehler DB Länge nicht ausreichend
      L     #Zeiger_Ziel;
      L     DW#16#FFFFFF;
      AD;
      L     W#16#85;
      CAD;
      +D;
      T     #Zeiger_Ziel;
ZNDB: NOP   0;
NETWORK
TITLE = Bytes kopieren
//geschwindigkeitsopitmiert:
//- Schleifenzäehler bleibt in AKKU1 und AKKU2
//- Kopieren über Worte, letztes Byte (ungerade Bytezahl) separat.
// (network holds code this reader does not know; not shown)
NETWORK
TITLE = Fehlerauswertung
      L     0;	//kein Fehler
      JU    SEFE;	//  setze Fehlerausgang
      L     -1;	//Bereichszeiger Quelle falsch
      JU    SEFE;	//  setze Fehlerausgang
      L     -2;	//Bereichszeiger Ziel falsch
      JU    SEFE;	//  setze Fehlerausgang
BLFE: L     -3;	//Blocklänge falsch
      JU    SEFE;	//  setze Fehlerausgang
DBNX: L     -4;	//Datenbaustein nicht existent 
      JU    SEFE;	//  setze Fehlerausgang
DBLF: L     -5;	//Datenbaustein Längenfehler
      JU    SEFE;	//  setze Fehlerausgang
DTFE: L     -6;	//Fehler Datentyp in ANY-Zeiger
      JU    SEFE;	//  setze Fehlerausgang         (004)
      L     -7;	//Fehler Anfangsbyte negativ    (004)
SEFE: T     #out_Fehler;
NETWORK
TITLE = DB-Register wiederherstellen
      OPN   DB [#G_DB_SAVE];
      OPN   DI [#I_DB_SAVE];
NETWORK
TITLE = BIE-Bit zuweisen
      L     #out_Fehler;
      L     0;
      ==I;
      SAVE;
END_FUNCTION

